// TIA Portal project "2025-26_Estampadora_Botonera_V17" (V17)

(* hardware
DEVICE "S7-1200 station_1"  S7-1200 Station
   slot 0: "Rack_0"  S7-1200 Rack  Rack  V1.0
   slot 1: "PLC_1"  CPU 1214C AC/DC/Rly  6ES7 214-1BG40-0XB0  V4.5
   slot 3: "AQ 1x12BIT_1"  AQ1 signal board  6ES7 232-4HA30-0XB0  V1.0
DEVICE "HMI_1"  KTP700 Basic PN
   slot 0: "HMI_1"  KTP700 Basic PN  6AV2 123-2GB03-0AX0  17.0.0.0
   slot 1: "HMI_RT_1"  KTP700 Basic PN  6AV2 123-2GB03-0AX0  17.0.0.0
   slot 5: "HMI_1.IE_CP_1"  PROFINET Interface  17.0.0.0
      slot 1: "PROFINET Interface_1"  PROFINET Interface
         slot 1: "Port_1"  Port
*)

// ===== PLC "PLC_1"  CPU 1214C AC/DC/Rly =====

VAR_GLOBAL   // PLC tag table "Tabla de variables estándar"
   "System_Byte" AT %MB1000 : Byte;
   "FirstScan" AT %M1000.0 : Bool;
   "DiagStatusUpdate" AT %M1000.1 : Bool;
   "AlwaysTRUE" AT %M1000.2 : Bool;
   "AlwaysFALSE" AT %M1000.3 : Bool;
   "INTERNA_Vacuna_libre" AT %M1001.0 : Bool;
   "INTERNA_Embalando_vacuna" AT %M1001.1 : Bool;
   "INTERNA_Soporte_libre" AT %M1001.2 : Bool;
   "INTERNA_Embalando_soporte" AT %M1001.3 : Bool;
   "INTERNA_Caja_libre" AT %M1001.4 : Bool;
   "INTERNA_Embalando_caja" AT %M1001.5 : Bool;
   "INTERNA_Robot_libre" AT %M1001.6 : Bool;
   "INTERNA_Robot_vacuna_hecho" AT %M1001.7 : Bool;
   "INTERNA_Robot_soporte_hecho" AT %M1002.0 : Bool;
   "OPCIN_sensor_caja_2" AT %I2.1 : Bool;
   "OPCIN_sensor_caja_1" AT %I2.0 : Bool;
   "OPCIN_sensor_caja_3" AT %I2.2 : Bool;
   "OPCIN_sensor_caja_A" AT %I2.3 : Bool;
   "OPCIN_sensor_caja_B" AT %I2.5 : Bool;
   "OPCIN_Emp_caja_A_front" AT %I3.1 : Bool;
   "OPCIN_Emp_caja_A_back" AT %I2.6 : Bool;
   "OPCIN_Emp_caja_B_front" AT %I2.7 : Bool;
   "OPCIN_Emp_caja_B_back" AT %I3.0 : Bool;
   "OPCOUT_Cinta_pre_caja" AT %Q2.0 : Bool;
   "OPCOUT_Cinta_post_caja" AT %Q2.1 : Bool;
   "OPCOUT_Cinta_alma_caja" AT %Q2.4 : Bool;
   "OPCOUT_Emp_caja_A" AT %Q2.2 : Bool;
   "OPCOUT_Emp_caja_B" AT %Q2.3 : Bool;
   "OPCOUT_Cajas" AT %Q3.2 : Bool;
   "OPCIN_Sensor_soporte" AT %I1.0 : Bool;
   "OPCIN_Vision_soporte" AT %IW34 : Int;
   "OPCIN_Sensor_soporte_A" AT %I1.2 : Bool;
   "OPCIN_Sensor_soporte_B" AT %I1.1 : Bool;
   "OPCIN_Emp_soporte_A_front" AT %I1.7 : Bool;
   "OPCIN_Emp_soporte_A_back" AT %I1.6 : Bool;
   "OPCIN_Emp_soporte_B_front" AT %I1.5 : Bool;
   "OPCIN_Emp_soporte_B_back" AT %I1.4 : Bool;
   "OPCOUT_Cinta_pre_soporte" AT %Q1.0 : Bool;
   "OPCOUT_Cinta_post_soporte" AT %Q1.1 : Bool;
   "OPCOUT_Cinta_alma_soporte" AT %Q1.5 : Bool;
   "OPCOUT_Cinta_curva_soporte" AT %Q1.4 : Bool;
   "OPCOUT_Soporte" AT %Q3.1 : Bool;
   "OPCOUT_Emp_soporte_A" AT %Q1.3 : Bool;
   "OPCOUT_Emp_soporte_B" AT %Q1.2 : Bool;
   "OPCIN_Sensor_vacuna" AT %I0.0 : Bool;
   "OPCIN_Vision_vacuna" AT %IW30 : Int;
   "OPCIN_Sensor_vacuna_A" AT %I0.2 : Bool;
   "OPCIN_Sensor_vacuna_B" AT %I0.1 : Bool;
   "OPCIN_Emp_vacuna_B_front" AT %I0.5 : Bool;
   "OPCIN_Emp_vacuna_B_back" AT %I0.4 : Bool;
   "OPCIN_Emp_vacuna_A_front" AT %I0.7 : Bool;
   "OPCIN_Emp_vacuna_A_back" AT %I0.6 : Bool;
   "OPCOUT_Cinta_pre_vacunas" AT %Q0.0 : Bool;
   "OPCOUT_Vacunas" AT %Q3.0 : Bool;
   "OPCOUT_Cinta_post_vacuna" AT %Q0.1 : Bool;
   "OPCOUT_Emp_vacuna_B" AT %Q0.2 : Bool;
   "OPCOUT_Emp_vacuna_A" AT %Q0.3 : Bool;
   "OPCOUT_Cinta_alma_vacuna" AT %Q0.5 : Bool;
   "OPCOUT_Cinta_curva_vacuna" AT %Q0.4 : Bool;
   "OPCIN_sensor_alma_soporte" AT %I1.3 : Bool;
   "OPCIN_sensor_alma_vacuna" AT %I0.3 : Bool;
   "OPCIN_sensor_alma_caja" AT %I2.4 : Bool;
   "OPCIN_PP_Rotating" AT %I3.5 : Bool;
   "OPCIN_PP_Moving_X" AT %I3.3 : Bool;
   "OPCIN_PP_Detected" AT %I3.2 : Bool;
   "OPCIN_PP_Moving_Z" AT %I3.4 : Bool;
   "OPCOUT_PP_CW" AT %Q3.4 : Bool;
   "OPCOUT_PP_CCW" AT %Q3.5 : Bool;
   "OPCOUT_PP_X" AT %Q3.6 : Bool;
   "OPCOUT_PP_Z" AT %Q3.7 : Bool;
   "OPCOUT_PP_Grab" AT %Q3.3 : Bool;
   "INTERNA_Robot_soporte" AT %M1002.1 : Bool;
   "INTERNA_Robot_vacuna" AT %M1002.2 : Bool;
   "CW_ROB1" AT %M1002.3 : Bool;
   "CW_ROB2" AT %M1002.4 : Bool;
   "CCW_ROB1" AT %M1002.5 : Bool;
   "CCW_ROB2" AT %M1002.6 : Bool;
   "GRAB_ROB1" AT %M1002.7 : Bool;
   "GRAB_ROB2" AT %M1003.0 : Bool;
   "X_ROB1" AT %M1003.1 : Bool;
   "X_ROB2" AT %M1003.2 : Bool;
   "Z_ROB1" AT %M1003.3 : Bool;
   "Z_ROB2" AT %M1003.4 : Bool;
   "CIN_ALMA_1" AT %M1003.5 : Bool;
   "CIN_ALMA_2" AT %M1003.6 : Bool;
   "Alarma_vacuna" AT %M1003.7 : Bool;
   "Alarma_soporte" AT %M1004.0 : Bool;
   "Alarma_caja" AT %M1004.1 : Bool;
   "BOOL_EMERGENCIA" AT %M1004.2 : Bool;
   "BOOL_REARME" AT %M1004.3 : Bool;
   "OPCIN_RESET" AT %I4.0 : Bool;
   "OPCIN_RESUME" AT %I4.1 : Bool;
   "OPCIN_SALIDA" AT %I4.2 : Bool;
   "OPCOUT_N_CICLOS" AT %QW30 : Int;
   "OPCIN_SETA" AT %I4.3 : Bool;
   "RESET" AT %M1004.4 : Bool;
   "RESUME" AT %M1004.5 : Bool;
   "FINAL" AT %M1004.6 : Bool;
   "SETA" AT %M1004.7 : Bool;
END_VAR

DATA_BLOCK "Llamadas_Robot_DB"   // DB4
{ S7_Optimized_Access := 'TRUE' }
VERSION : 0.1
// stored: InstanceOfName HANDLER
"HANDLER"
BEGIN
END_DATA_BLOCK

DATA_BLOCK "DATOS_HMI"   // DB18
{ S7_Optimized_Access := 'TRUE' }
VERSION : 0.1
   VAR
      Boton_Reset : Bool;
      Boton_Resume : Bool;
      Estado_Alarma : Bool;
      Estado_Vacuna : Int;
      Estado_Soporte : Int;
      Estado_Caja : Int;
      Estado_Embalaje : Int;
      "CAJAS TOTALES" : Int;
      "SETA EMERGENCIA" : Bool;
      "BOTON REARME" : Bool;
      "FIN DE PISTA" : Bool;
   END_VAR
BEGIN
END_DATA_BLOCK

DATA_BLOCK "EMERGENCIA_DB"   // DB19
{ S7_Optimized_Access := 'TRUE' }
VERSION : 0.1
// stored: InstanceOfName EMERGENCIA
"EMERGENCIA"
BEGIN
END_DATA_BLOCK

DATA_BLOCK "Cinta_Vacunas_DB"   // DB34
{ S7_Optimized_Access := 'TRUE' }
VERSION : 0.1
// stored: InstanceOfName Cinta_Vacunas
"Cinta_Vacunas"
BEGIN
END_DATA_BLOCK

DATA_BLOCK "Cinta_Vacunas_DB_1"   // DB49
{ S7_Optimized_Access := 'TRUE' }
VERSION : 0.1
// stored: InstanceOfName Cinta_Vacunas
"Cinta_Vacunas"
BEGIN
END_DATA_BLOCK

DATA_BLOCK "Cinta_soporte_DB"   // DB50
{ S7_Optimized_Access := 'TRUE' }
VERSION : 0.1
// stored: InstanceOfName Cinta_soporte
"Cinta_soporte"
BEGIN
END_DATA_BLOCK

DATA_BLOCK "Cinta_soporte_DB_1"   // DB51
{ S7_Optimized_Access := 'TRUE' }
VERSION : 0.1
// stored: InstanceOfName Cinta_soporte
"Cinta_soporte"
BEGIN
END_DATA_BLOCK

DATA_BLOCK "Cinta_cajas_DB"   // DB52
{ S7_Optimized_Access := 'TRUE' }
VERSION : 0.1
// stored: InstanceOfName Cinta_cajas
"Cinta_cajas"
BEGIN
END_DATA_BLOCK

DATA_BLOCK "Embalaje_DB"   // DB53
{ S7_Optimized_Access := 'TRUE' }
VERSION : 0.1
// stored: InstanceOfName Embalaje
"Embalaje"
BEGIN
END_DATA_BLOCK

DATA_BLOCK "Robot_Vacuna_DB"   // DB54
{ S7_Optimized_Access := 'TRUE' }
VERSION : 0.1
// stored: InstanceOfName Robot_Vacuna
"Robot_Vacuna"
BEGIN
END_DATA_BLOCK

DATA_BLOCK "Robot_Soporte_DB"   // DB55
{ S7_Optimized_Access := 'TRUE' }
VERSION : 0.1
// stored: InstanceOfName Robot_Soporte
"Robot_Soporte"
BEGIN
END_DATA_BLOCK

// folder: System blocks/Program resources

DATA_BLOCK "2s/X41"   // DB1
{ S7_Optimized_Access := 'TRUE' }
AUTHOR : Simatic
FAMILY : IEC
NAME : IEC_TMR
VERSION : 1.0
// stored: InstanceOfName IEC_TIMER
"IEC_TIMER"
BEGIN
END_DATA_BLOCK

DATA_BLOCK "2s/x42"   // DB2
{ S7_Optimized_Access := 'TRUE' }
AUTHOR : Simatic
FAMILY : IEC
NAME : IEC_TMR
VERSION : 1.0
// stored: InstanceOfName IEC_TIMER
"IEC_TIMER"
BEGIN
END_DATA_BLOCK

DATA_BLOCK "2s/X34"   // DB3
{ S7_Optimized_Access := 'TRUE' }
AUTHOR : Simatic
FAMILY : IEC
NAME : IEC_TMR
VERSION : 1.0
// stored: InstanceOfName IEC_TIMER
"IEC_TIMER"
BEGIN
END_DATA_BLOCK

DATA_BLOCK "T_Alarma_2"   // DB5
{ S7_Optimized_Access := 'TRUE' }
AUTHOR : Simatic
FAMILY : IEC
NAME : IEC_TMR
VERSION : 1.0
// stored: InstanceOfName IEC_TIMER
"IEC_TIMER"
BEGIN
END_DATA_BLOCK

DATA_BLOCK "T_Alarma_5"   // DB6
{ S7_Optimized_Access := 'TRUE' }
AUTHOR : Simatic
FAMILY : IEC
NAME : IEC_TMR
VERSION : 1.0
// stored: InstanceOfName IEC_TIMER
"IEC_TIMER"
BEGIN
END_DATA_BLOCK

DATA_BLOCK "T_Alarma_7"   // DB7
{ S7_Optimized_Access := 'TRUE' }
AUTHOR : Simatic
FAMILY : IEC
NAME : IEC_TMR
VERSION : 1.0
// stored: InstanceOfName IEC_TIMER
"IEC_TIMER"
BEGIN
END_DATA_BLOCK

DATA_BLOCK "T_Alarma_7_PRIMA"   // DB8
{ S7_Optimized_Access := 'TRUE' }
AUTHOR : Simatic
FAMILY : IEC
NAME : IEC_TMR
VERSION : 1.0
// stored: InstanceOfName IEC_TIMER
"IEC_TIMER"
BEGIN
END_DATA_BLOCK

DATA_BLOCK "T_Alarma_3"   // DB9
{ S7_Optimized_Access := 'TRUE' }
AUTHOR : Simatic
FAMILY : IEC
NAME : IEC_TMR
VERSION : 1.0
// stored: InstanceOfName IEC_TIMER
"IEC_TIMER"
BEGIN
END_DATA_BLOCK

DATA_BLOCK "T_alarma_6"   // DB10
{ S7_Optimized_Access := 'TRUE' }
AUTHOR : Simatic
FAMILY : IEC
NAME : IEC_TMR
VERSION : 1.0
// stored: InstanceOfName IEC_TIMER
"IEC_TIMER"
BEGIN
END_DATA_BLOCK

DATA_BLOCK "T_Alarma_9"   // DB11
{ S7_Optimized_Access := 'TRUE' }
AUTHOR : Simatic
FAMILY : IEC
NAME : IEC_TMR
VERSION : 1.0
// stored: InstanceOfName IEC_TIMER
"IEC_TIMER"
BEGIN
END_DATA_BLOCK

DATA_BLOCK "T_Alarma_9_PRIMA"   // DB12
{ S7_Optimized_Access := 'TRUE' }
AUTHOR : Simatic
FAMILY : IEC
NAME : IEC_TMR
VERSION : 1.0
// stored: InstanceOfName IEC_TIMER
"IEC_TIMER"
BEGIN
END_DATA_BLOCK

DATA_BLOCK "TIMER_ALARMA_FRESADORA"   // DB13
{ S7_Optimized_Access := 'TRUE' }
AUTHOR : Simatic
FAMILY : IEC
NAME : IEC_TMR
VERSION : 1.0
// stored: InstanceOfName IEC_TIMER
"IEC_TIMER"
BEGIN
END_DATA_BLOCK

DATA_BLOCK "T_alarma_1"   // DB14
{ S7_Optimized_Access := 'TRUE' }
AUTHOR : Simatic
FAMILY : IEC
NAME : IEC_TMR
VERSION : 1.0
// stored: InstanceOfName IEC_TIMER
"IEC_TIMER"
BEGIN
END_DATA_BLOCK

DATA_BLOCK "T_alarma_4"   // DB15
{ S7_Optimized_Access := 'TRUE' }
AUTHOR : Simatic
FAMILY : IEC
NAME : IEC_TMR
VERSION : 1.0
// stored: InstanceOfName IEC_TIMER
"IEC_TIMER"
BEGIN
END_DATA_BLOCK

DATA_BLOCK "T_alarma_8"   // DB16
{ S7_Optimized_Access := 'TRUE' }
AUTHOR : Simatic
FAMILY : IEC
NAME : IEC_TMR
VERSION : 1.0
// stored: InstanceOfName IEC_TIMER
"IEC_TIMER"
BEGIN
END_DATA_BLOCK

DATA_BLOCK "T_alarma_8_PRIMA"   // DB17
{ S7_Optimized_Access := 'TRUE' }
AUTHOR : Simatic
FAMILY : IEC
NAME : IEC_TMR
VERSION : 1.0
// stored: InstanceOfName IEC_TIMER
"IEC_TIMER"
BEGIN
END_DATA_BLOCK

DATA_BLOCK "1S/X411"   // DB20
{ S7_Optimized_Access := 'TRUE' }
AUTHOR : Simatic
FAMILY : IEC
NAME : IEC_TMR
VERSION : 1.0
// stored: InstanceOfName IEC_TIMER
"IEC_TIMER"
BEGIN
END_DATA_BLOCK

DATA_BLOCK "Timer_1s_X04A"   // DB21
{ S7_Optimized_Access := 'TRUE' }
AUTHOR : Simatic
FAMILY : IEC
NAME : IEC_TMR
VERSION : 1.0
// stored: InstanceOfName IEC_TIMER
"IEC_TIMER"
BEGIN
END_DATA_BLOCK

DATA_BLOCK "Timer_1s_X03"   // DB22
{ S7_Optimized_Access := 'TRUE' }
AUTHOR : Simatic
FAMILY : IEC
NAME : IEC_TMR
VERSION : 1.0
// stored: InstanceOfName IEC_TIMER
"IEC_TIMER"
BEGIN
END_DATA_BLOCK

DATA_BLOCK "Timer_1s_X130A"   // DB23
{ S7_Optimized_Access := 'TRUE' }
AUTHOR : Simatic
FAMILY : IEC
NAME : IEC_TMR
VERSION : 1.0
// stored: InstanceOfName IEC_TIMER
"IEC_TIMER"
BEGIN
END_DATA_BLOCK

DATA_BLOCK "Timer_1s_X130B"   // DB24
{ S7_Optimized_Access := 'TRUE' }
AUTHOR : Simatic
FAMILY : IEC
NAME : IEC_TMR
VERSION : 1.0
// stored: InstanceOfName IEC_TIMER
"IEC_TIMER"
BEGIN
END_DATA_BLOCK

DATA_BLOCK "1s/X231A"   // DB25
{ S7_Optimized_Access := 'TRUE' }
AUTHOR : Simatic
FAMILY : IEC
NAME : IEC_TMR
VERSION : 1.0
// stored: InstanceOfName IEC_TIMER
"IEC_TIMER"
BEGIN
END_DATA_BLOCK

DATA_BLOCK "1s/X230B"   // DB26
{ S7_Optimized_Access := 'TRUE' }
AUTHOR : Simatic
FAMILY : IEC
NAME : IEC_TMR
VERSION : 1.0
// stored: InstanceOfName IEC_TIMER
"IEC_TIMER"
BEGIN
END_DATA_BLOCK

DATA_BLOCK "1S/X230C"   // DB27
{ S7_Optimized_Access := 'TRUE' }
AUTHOR : Simatic
FAMILY : IEC
NAME : IEC_TMR
VERSION : 1.0
// stored: InstanceOfName IEC_TIMER
"IEC_TIMER"
BEGIN
END_DATA_BLOCK

DATA_BLOCK "3s/x37"   // DB28
{ S7_Optimized_Access := 'TRUE' }
AUTHOR : Simatic
FAMILY : IEC
NAME : IEC_TMR
VERSION : 1.0
// stored: InstanceOfName IEC_TIMER
"IEC_TIMER"
BEGIN
END_DATA_BLOCK

DATA_BLOCK "1s/X311B"   // DB29
{ S7_Optimized_Access := 'TRUE' }
AUTHOR : Simatic
FAMILY : IEC
NAME : IEC_TMR
VERSION : 1.0
// stored: InstanceOfName IEC_TIMER
"IEC_TIMER"
BEGIN
END_DATA_BLOCK

DATA_BLOCK "1s/X311C"   // DB30
{ S7_Optimized_Access := 'TRUE' }
AUTHOR : Simatic
FAMILY : IEC
NAME : IEC_TMR
VERSION : 1.0
// stored: InstanceOfName IEC_TIMER
"IEC_TIMER"
BEGIN
END_DATA_BLOCK

DATA_BLOCK "1s/X321A"   // DB31
{ S7_Optimized_Access := 'TRUE' }
AUTHOR : Simatic
FAMILY : IEC
NAME : IEC_TMR
VERSION : 1.0
// stored: InstanceOfName IEC_TIMER
"IEC_TIMER"
BEGIN
END_DATA_BLOCK

DATA_BLOCK "1S/X311"   // DB32
{ S7_Optimized_Access := 'TRUE' }
AUTHOR : Simatic
FAMILY : IEC
NAME : IEC_TMR
VERSION : 1.0
// stored: InstanceOfName IEC_TIMER
"IEC_TIMER"
BEGIN
END_DATA_BLOCK

DATA_BLOCK "1s/X39"   // DB33
{ S7_Optimized_Access := 'TRUE' }
AUTHOR : Simatic
FAMILY : IEC
NAME : IEC_TMR
VERSION : 1.0
// stored: InstanceOfName IEC_TIMER
"IEC_TIMER"
BEGIN
END_DATA_BLOCK

DATA_BLOCK "1s/X410"   // DB35
{ S7_Optimized_Access := 'TRUE' }
AUTHOR : Simatic
FAMILY : IEC
NAME : IEC_TMR
VERSION : 1.0
// stored: InstanceOfName IEC_TIMER
"IEC_TIMER"
BEGIN
END_DATA_BLOCK

DATA_BLOCK "1s/X44"   // DB36
{ S7_Optimized_Access := 'TRUE' }
AUTHOR : Simatic
FAMILY : IEC
NAME : IEC_TMR
VERSION : 1.0
// stored: InstanceOfName IEC_TIMER
"IEC_TIMER"
BEGIN
END_DATA_BLOCK

DATA_BLOCK "2s/X45"   // DB37
{ S7_Optimized_Access := 'TRUE' }
AUTHOR : Simatic
FAMILY : IEC
NAME : IEC_TMR
VERSION : 1.0
// stored: InstanceOfName IEC_TIMER
"IEC_TIMER"
BEGIN
END_DATA_BLOCK

DATA_BLOCK "2s/X46"   // DB38
{ S7_Optimized_Access := 'TRUE' }
AUTHOR : Simatic
FAMILY : IEC
NAME : IEC_TMR
VERSION : 1.0
// stored: InstanceOfName IEC_TIMER
"IEC_TIMER"
BEGIN
END_DATA_BLOCK

DATA_BLOCK "1s/X47"   // DB39
{ S7_Optimized_Access := 'TRUE' }
AUTHOR : Simatic
FAMILY : IEC
NAME : IEC_TMR
VERSION : 1.0
// stored: InstanceOfName IEC_TIMER
"IEC_TIMER"
BEGIN
END_DATA_BLOCK

DATA_BLOCK "1s/X48"   // DB40
{ S7_Optimized_Access := 'TRUE' }
AUTHOR : Simatic
FAMILY : IEC
NAME : IEC_TMR
VERSION : 1.0
// stored: InstanceOfName IEC_TIMER
"IEC_TIMER"
BEGIN
END_DATA_BLOCK

DATA_BLOCK "1s/X49"   // DB41
{ S7_Optimized_Access := 'TRUE' }
AUTHOR : Simatic
FAMILY : IEC
NAME : IEC_TMR
VERSION : 1.0
// stored: InstanceOfName IEC_TIMER
"IEC_TIMER"
BEGIN
END_DATA_BLOCK

DATA_BLOCK "1S/X511"   // DB42
{ S7_Optimized_Access := 'TRUE' }
AUTHOR : Simatic
FAMILY : IEC
NAME : IEC_TMR
VERSION : 1.0
// stored: InstanceOfName IEC_TIMER
"IEC_TIMER"
BEGIN
END_DATA_BLOCK

DATA_BLOCK "1S/X54"   // DB43
{ S7_Optimized_Access := 'TRUE' }
AUTHOR : Simatic
FAMILY : IEC
NAME : IEC_TMR
VERSION : 1.0
// stored: InstanceOfName IEC_TIMER
"IEC_TIMER"
BEGIN
END_DATA_BLOCK

DATA_BLOCK "2S/X55"   // DB44
{ S7_Optimized_Access := 'TRUE' }
AUTHOR : Simatic
FAMILY : IEC
NAME : IEC_TMR
VERSION : 1.0
// stored: InstanceOfName IEC_TIMER
"IEC_TIMER"
BEGIN
END_DATA_BLOCK

DATA_BLOCK "2S/X56"   // DB45
{ S7_Optimized_Access := 'TRUE' }
AUTHOR : Simatic
FAMILY : IEC
NAME : IEC_TMR
VERSION : 1.0
// stored: InstanceOfName IEC_TIMER
"IEC_TIMER"
BEGIN
END_DATA_BLOCK

DATA_BLOCK "2S/X57"   // DB46
{ S7_Optimized_Access := 'TRUE' }
AUTHOR : Simatic
FAMILY : IEC
NAME : IEC_TMR
VERSION : 1.0
// stored: InstanceOfName IEC_TIMER
"IEC_TIMER"
BEGIN
END_DATA_BLOCK

DATA_BLOCK "1S/X59"   // DB47
{ S7_Optimized_Access := 'TRUE' }
AUTHOR : Simatic
FAMILY : IEC
NAME : IEC_TMR
VERSION : 1.0
// stored: InstanceOfName IEC_TIMER
"IEC_TIMER"
BEGIN
END_DATA_BLOCK

DATA_BLOCK "2S/X510"   // DB48
{ S7_Optimized_Access := 'TRUE' }
AUTHOR : Simatic
FAMILY : IEC
NAME : IEC_TMR
VERSION : 1.0
// stored: InstanceOfName IEC_TIMER
"IEC_TIMER"
BEGIN
END_DATA_BLOCK

DATA_BLOCK "1S/X8.5"   // DB56
{ S7_Optimized_Access := 'TRUE' }
AUTHOR : Simatic
FAMILY : IEC
NAME : IEC_TMR
VERSION : 1.0
// stored: InstanceOfName IEC_TIMER
"IEC_TIMER"
BEGIN
END_DATA_BLOCK

DATA_BLOCK "XAUX"   // DB57
{ S7_Optimized_Access := 'TRUE' }
AUTHOR : Simatic
FAMILY : IEC
NAME : IEC_TMR
VERSION : 1.0
// stored: InstanceOfName IEC_TIMER
"IEC_TIMER"
BEGIN
END_DATA_BLOCK

DATA_BLOCK "2S/XAUX2"   // DB58
{ S7_Optimized_Access := 'TRUE' }
AUTHOR : Simatic
FAMILY : IEC
NAME : IEC_TMR
VERSION : 1.0
// stored: InstanceOfName IEC_TIMER
"IEC_TIMER"
BEGIN
END_DATA_BLOCK

DATA_BLOCK "1S/X412"   // DB59
{ S7_Optimized_Access := 'TRUE' }
AUTHOR : Simatic
FAMILY : IEC
NAME : IEC_TMR
VERSION : 1.0
// stored: InstanceOfName IEC_TIMER
"IEC_TIMER"
BEGIN
END_DATA_BLOCK

DATA_BLOCK "2S/X511"   // DB60
{ S7_Optimized_Access := 'TRUE' }
AUTHOR : Simatic
FAMILY : IEC
NAME : IEC_TMR
VERSION : 1.0
// stored: InstanceOfName IEC_TIMER
"IEC_TIMER"
BEGIN
END_DATA_BLOCK

DATA_BLOCK "2S/X512"   // DB61
{ S7_Optimized_Access := 'TRUE' }
AUTHOR : Simatic
FAMILY : IEC
NAME : IEC_TMR
VERSION : 1.0
// stored: InstanceOfName IEC_TIMER
"IEC_TIMER"
BEGIN
END_DATA_BLOCK

DATA_BLOCK "2S/X513"   // DB62
{ S7_Optimized_Access := 'TRUE' }
AUTHOR : Simatic
FAMILY : IEC
NAME : IEC_TMR
VERSION : 1.0
// stored: InstanceOfName IEC_TIMER
"IEC_TIMER"
BEGIN
END_DATA_BLOCK

DATA_BLOCK "2S/X514"   // DB63
{ S7_Optimized_Access := 'TRUE' }
AUTHOR : Simatic
FAMILY : IEC
NAME : IEC_TMR
VERSION : 1.0
// stored: InstanceOfName IEC_TIMER
"IEC_TIMER"
BEGIN
END_DATA_BLOCK

DATA_BLOCK "2S/X58"   // DB64
{ S7_Optimized_Access := 'TRUE' }
AUTHOR : Simatic
FAMILY : IEC
NAME : IEC_TMR
VERSION : 1.0
// stored: InstanceOfName IEC_TIMER
"IEC_TIMER"
BEGIN
END_DATA_BLOCK

DATA_BLOCK "2S/X52"   // DB65
{ S7_Optimized_Access := 'TRUE' }
AUTHOR : Simatic
FAMILY : IEC
NAME : IEC_TMR
VERSION : 1.0
// stored: InstanceOfName IEC_TIMER
"IEC_TIMER"
BEGIN
END_DATA_BLOCK

// folder: (top level)

FUNCTION_BLOCK "Embalaje"   // FB1, SCL
{ S7_Optimized_Access := 'TRUE' }
VERSION : 0.1
   VAR_INPUT
      sensor_alma_soporte : Bool;
      sensor_alma_vacuna : Bool;
      sensor_alma_caja_1 : Bool;
      Robot_libre : Bool;
      Robot_soporte_hecho : Bool;
      Robot_vacuna_hecho : Bool;
      N_soportes : Int := 1;
      N_vacunas : Int := 1;
      EMERGENCIA : Bool;
      REARME : Bool;
      "FIN DE PISTA" : Bool;
   END_VAR
   VAR_OUTPUT
      N_ESTADO : Int;
      Soporte_libre : Bool;
      Vacuna_libre : Bool;
      Embalando_soporte : Bool;
      Embalando_vacuna : Bool;
      Caja_libre : Bool;
      Embalando_caja : Bool;
      Robot_soporte : Bool;
      Robot_vacuna : Bool;
      Cinta_alma_caja : Bool;
      CAJAS_TOTALES : Int;
   END_VAR
   VAR
      Flanco_x35 : R_TRIG;
      Flanco_x36 : R_TRIG;
      Flanco_X37 : R_TRIG;
      Count_soportes : Int;
      Count_vacunas : Int;
      X30 : Bool;
      X310A : Bool;
      X310B : Bool;
      X311B : Bool;
      X310C : Bool;
      X311C : Bool;
      X320A : Bool;
      X321A : Bool;
      X320B : Bool;
      X33 : Bool;
      X34 : Bool;
      X35 : Bool;
      X36 : Bool;
      X37 : Bool;
      X38 : Bool;
      X39 : Bool;
      X310 : Bool;
      X311 : Bool;
      S30 : Bool;
      S310A : Bool;
      S310B : Bool;
      S311B : Bool;
      S310C : Bool;
      S311C : Bool;
      S320A : Bool;
      S321A : Bool;
      S320B : Bool;
      S33 : Bool;
      S34 : Bool;
      S35 : Bool;
      S36 : Bool;
      S37 : Bool;
      S38 : Bool;
      S39 : Bool;
      S310 : Bool;
      S311 : Bool;
   END_VAR
BEGIN
   "3s/x37".TON(IN:=#X37,
                PT:=T#3s);
   "1s/X311B".TON(IN:=#X311B,
                  PT:=T#1s);
   "1s/X311C".TON(IN:=#X311C,
                  PT:=T#1s);
   "1s/X321A".TON(IN:=#X321A,
                  PT:=T#1s);
   "1S/X311".TON(IN:=#X311,
                 PT:=T#1s);
   "1s/X39".TON(IN:=#X39,
                PT:=t#1s);
   "2s/X34".TON(IN:=#X34,
                PT:=T#2S);

   IF NOT #EMERGENCIA THEN
       //FUNCIONES DE TRANSICIÓN
       #S30 := (#X37 AND "3s/x37".Q) OR (#X311B) OR (#X311C) OR "FirstScan";
       IF NOT #"FIN DE PISTA" THEN
           #S310A := #X30 AND #sensor_alma_soporte AND #sensor_alma_vacuna;
           #S310B := #X30 AND NOT #sensor_alma_soporte;
           #S310C := #X30 AND NOT #sensor_alma_vacuna;
       ELSE
           #S310A := FALSE;
           #S310B := FALSE;
           #S310C := FALSE;
       END_IF;
       #S311B := #X310B AND #sensor_alma_soporte;
       #S311C := #X310C AND #sensor_alma_vacuna;
       #S320A := #X310A AND NOT #sensor_alma_caja_1;
       #S321A := #X320A AND #sensor_alma_caja_1;
       #S320B := #X320A AND #sensor_alma_caja_1;
       #S33 := (#X321A AND "1s/X321A".Q) OR #X320B;
       #S34 := (#X33 AND #Robot_libre) OR (#X311 AND "1S/X311".Q);
       #S35 := (#X34 AND #Robot_vacuna_hecho AND "2s/X34".Q) OR (#X39);
       #S36 := #X35 AND (#Count_vacunas >= #N_vacunas) AND #Robot_soporte_hecho;
       #S37 := #X36 AND (#Count_soportes >= #N_soportes);
       #S38 := #X35 AND (#Count_vacunas < #N_vacunas) AND #Robot_soporte_hecho;
       #S39 := #X38 AND #sensor_alma_vacuna;
       #S310 := #X36 AND (#Count_soportes < #N_soportes);
       #S311 := #X310 AND #sensor_alma_soporte;

       //FUNCIONES DE ACTIVACIÓN DE ETAPAS
       #X30 := #S30 OR #X30 AND NOT (#S310A OR #S310B OR #S310C);
       #X310A := #S310A OR #X310A AND NOT (#S320A OR #S320B);
       #X320A := #S320A OR #X320A AND NOT #S321A;
       #X321A := #S321A OR #X321A AND NOT #S33;
       #X320B := #S320B OR #X320B AND NOT #S33;
       #X310B := #S310B OR #X310B AND NOT #S311B;
       #X311B := #S311B OR #X311B AND NOT #S30;
       #X310C := #S310C OR #X310C AND NOT #S311C;
       #X311C := #S311C OR #X311C AND NOT #S30;
       #X33 := #S33 OR #X33 AND NOT #S34;
       #X34 := #S34 OR #X34 AND NOT #S35;
       #X35 := #S35 OR #X35 AND NOT (#S36 OR #S38);
       #X36 := #S36 OR #X36 AND NOT (#S37 OR #S39);
       #X37 := #S37 OR #X37 AND NOT #S30;
       #X38 := #S38 OR #X38 AND NOT #S39;
       #X39 := #S39 OR #X39 AND NOT #S35;
       #X310 := #S310 OR #X310 AND NOT #S311;
       #X311 := #S311 OR #X311 AND NOT #S34;



       //FUNCIONES DE SALIDA
       #Soporte_libre := #X310B OR #X310;
       #Vacuna_libre := #X310C OR #X38;
       #Embalando_soporte := #X311B OR #X311;
       #Embalando_vacuna := #X311C OR #X39;
       #Caja_libre := #X320A;
       #Embalando_caja := #X321A;
       #Robot_soporte := #X35;
       #Robot_vacuna := #X34;
       #Cinta_alma_caja := #X37; 
   ELSE
       #Soporte_libre := FALSE;
       #Vacuna_libre := FALSE;
       #Embalando_soporte := FALSE;
       #Embalando_vacuna := FALSE;
       #Caja_libre := FALSE;
       #Embalando_caja := FALSE;
       #Robot_soporte := FALSE;
       #Robot_vacuna := FALSE;
       #Cinta_alma_caja := FALSE;

   END_IF;

   IF #REARME THEN
       #X30 := TRUE;
       #X310A := FALSE;
       #X320A := FALSE;
       #X321A := FALSE;
       #X320B := FALSE;
       #X310B := FALSE;
       #X311B := FALSE;
       #X310C := FALSE;
       #X311C := FALSE;
       #X33 := FALSE;
       #X34 := FALSE;
       #X35 := FALSE;
       #X36 := FALSE;
       #X37 := FALSE;
       #X38 := FALSE;
       #X39 := FALSE;
       #X310 := FALSE;
       #X311 := FALSE;
   END_IF;

   IF #X30 OR #X310A OR #X320B THEN
       #N_ESTADO := 0;
   ELSIF #X310B OR #X311B THEN
       #N_ESTADO := 1;
   ELSIF #X310C OR #X311C THEN
       #N_ESTADO := 2;
   ELSIF #X320A OR #X321A THEN
       #N_ESTADO := 3;
   ELSIF #X33 THEN
       #N_ESTADO := 4;
   ELSIF #X34 THEN
       #N_ESTADO := 5;
   ELSIF #X35 THEN
       #N_ESTADO := 6;
   ELSIF #X38 OR #X39 THEN
       #N_ESTADO := 7;
   ELSIF #X36 THEN
       #N_ESTADO := 8;
   ELSIF #X310 OR #X311 THEN
       #N_ESTADO := 9;
   ELSIF #X37 THEN
       #N_ESTADO := 10;
   END_IF;





   //CONTADORES
   #Flanco_x35(CLK := #X35);
   IF #Flanco_x35.Q THEN
       #Count_vacunas := #Count_vacunas + 1;
   END_IF;
   #Flanco_x36(CLK := #X36);
   IF #Flanco_x36.Q THEN
       #Count_vacunas := 0;
       #Count_soportes := #Count_soportes + 1;
   END_IF;
   #Flanco_X37(CLK := #X37);
   IF #Flanco_X37.Q THEN
       #Count_soportes := 0;
       #CAJAS_TOTALES := #CAJAS_TOTALES + 1;
   END_IF;
END_FUNCTION_BLOCK

FUNCTION_BLOCK "Robot_Vacuna"   // FB2, SCL
{ S7_Optimized_Access := 'TRUE' }
VERSION : 0.1
   VAR_INPUT
      Robot_vacuna : Bool;
      PP_Rotating : Bool;
      PP_Moving_X : Bool;
      PP_Detected : Bool;
      EMERGENCIA : Bool;
      REARME : Bool;
   END_VAR
   VAR_OUTPUT
      PP_CW : Bool;
      PP_CCW : Bool;
      Robot_libre : Bool;
      PP_X : Bool;
      PP_Z : Bool;
      PP_Grab : Bool;
      Robot_vacuna_hecho : Bool;
   END_VAR
   VAR
      X40 : Bool;
      X41 : Bool;
      X42 : Bool;
      X43 : Bool;
      X44 : Bool;
      X45 : Bool;
      X46 : Bool;
      X47 : Bool;
      X48 : Bool;
      X49 : Bool;
      X410 : Bool;
      X411 : Bool;
      S40 : Bool;
      S41 : Bool;
      S42 : Bool;
      S43 : Bool;
      S44 : Bool;
      S45 : Bool;
      S46 : Bool;
      S47 : Bool;
      S48 : Bool;
      S49 : Bool;
      S410 : Bool;
      S411 : Bool;
      "X8,5" : Bool;
      "S8,5" : Bool;
      XAUX : Bool;
      SAUX : Bool;
      SAUX2 : Bool;
      XAUX2 : Bool;
      S412 : Bool;
      X412 : Bool;
   END_VAR
BEGIN
   "1s/X410".TON(IN:=#X410,
                 PT:=T#1s);
   "1s/X44".TON(IN:=#X44,
                PT:=T#2s);
   "2s/X45".TON(IN:=#X45,
                PT:=T#2s);
   "2s/X46".TON(IN:=#X46,
                PT:=T#2s);
   "1s/X47".TON(IN:=#X47,
                PT:=T#2s);
   "1s/X48".TON(IN:=#X48,
                PT:=T#2s);
   "1s/X49".TON(IN:=#X49,
                PT:=T#2s);
   "2s/X41".TON(IN:=#X41,
                PT:=T#2s);
   "2s/x42".TON(IN:=#X42,
                PT:=t#2s);
   "1S/X411".TON(IN:=#X411,
                   PT:=t#2s);

   "1S/X8.5".TON(IN:=#"X8,5",
                 PT:=T#2s);

   "XAUX".TON(IN:=#XAUX,
              PT:=T#2S);
   "2S/XAUX2".TON(IN:=#XAUX2,
                  PT:=T#2S);
   "1S/X412".TON(IN:=#X412,
                 PT:=T#1S);



   IF NOT #EMERGENCIA THEN
       //FUNCIONES DE TRANSICIÓN
       #S40 := (#X412 AND "1S/X412".Q) OR "FirstScan";
       #S41 := #X40 AND #Robot_vacuna;
       #S42 := #X41 AND "2s/X41".Q;(*

   *)
       #S43 := #X42 AND "2s/x42".Q;
       #S44 := #X43 AND #PP_Detected;
       #S45 := #X44 AND "1s/X44".Q;
       #S46 := #X45 AND "2s/X45".Q;
       #S47 := #X46 AND "2s/X46".Q;
       #S48 := #X47 AND "1s/X47".Q;
       #SAUX2 := #X48 AND "1s/X48".Q;
       #"S8,5" := #XAUX2 AND "2S/XAUX2".Q;
       #SAUX := #"X8,5" AND "1S/X8.5".Q;
       #S49 := #XAUX AND "XAUX".Q;
       #S410 := #X49 AND "1s/X49".Q;
       #S411:= #X410 AND "1s/X410".Q;
       #S412 := #X411 AND "1S/X411".Q;


       //FUNCIONES DE ACTIVACIÓN
       #X40 := #S40 OR #X40 AND NOT #S41;
       #X41 := #S41 OR #X41 AND NOT #S42;
       #X42 := #S42 OR #X42 AND NOT #S43;
       #X43 := #S43 OR #X43 AND NOT #S44;
       #X44 := #S44 OR #X44 AND NOT #S45;
       #X45 := #S45 OR #X45 AND NOT #S46;
       #X46 := #S46 OR #X46 AND NOT #S47;
       #X47 := #S47 OR #X47 AND NOT #S48;
       #X48 := #S48 OR #X48 AND NOT #SAUX2;
       #XAUX2 := #SAUX2 OR #XAUX2 AND NOT #"S8,5";
       #"X8,5" := #"S8,5" OR #"X8,5" AND NOT #SAUX;
       #XAUX := #SAUX OR #XAUX AND NOT #S49;
       #X49 := #S49 OR #X49 AND NOT #S410;
       #X410 := #S410 OR #X410 AND NOT #S411;
       #X411 := #S411 OR #X411 AND NOT #S412;
       #X412 := #S412 OR #X412 AND NOT #S40;


       //FUNCIONES DE SALIDA
       #Robot_libre := #X40;
       #PP_CW := #X47 OR #X48 OR #"X8,5";
       #PP_CCW := #X41 OR #X411;
       #PP_X := #X43 OR #X44 OR #X45 OR #X42 OR #X49 OR #X410;
       #PP_Z := #X43 OR #X44 OR #X410;
       #PP_Grab := #X44 OR #XAUX2 OR #X45 OR #X46 OR #X47 OR #X48 OR #X49 OR #X410 OR #"X8,5" OR #XAUX;
       #Robot_vacuna_hecho := #X412;
   ELSE
       #Robot_libre := FALSE;
       #PP_CW := FALSE;
       #PP_CCW := FALSE;
       #PP_X := FALSE;
       #PP_Z := FALSE;
       #PP_Grab := FALSE;
       #Robot_vacuna_hecho := FALSE;
   END_IF;

   IF #REARME THEN
       #X40 := TRUE;
       #X41 := FALSE;
       #X42 := FALSE;
       #X43 := FALSE;
       #X44 := FALSE;
       #X45 := FALSE;
       #X46 := FALSE;
       #X47 := FALSE;
       #X48 := FALSE;
       #X49 := FALSE;
       #X410 := FALSE;
   END_IF;
END_FUNCTION_BLOCK

FUNCTION_BLOCK "Robot_Soporte"   // FB3, SCL
{ S7_Optimized_Access := 'TRUE' }
VERSION : 0.1
   VAR_INPUT
      Robot_soporte : Bool;
      PP_Rotating : Bool;
      PP_Moving_X : Bool;
      PP_Detected : Bool;
      PP_Moving_Z : Bool;
      EMERGENCIA : Bool;
      REARME : Bool;
   END_VAR
   VAR_OUTPUT
      Robot_libre : Bool;
      PP_CW : Bool;
      PP_CCW : Bool;
      PP_X : Bool;
      PP_Z : Bool;
      PP_Grab : Bool;
      Robot_soporte_hecho : Bool;
   END_VAR
   VAR
      X50 : Bool;
      X51 : Bool;
      X52 : Bool;
      X53 : Bool;
      X54 : Bool;
      X55 : Bool;
      X56 : Bool;
      X57 : Bool;
      X58 : Bool;
      X59 : Bool;
      X510 : Bool;
      X511 : Bool;
      X512 : Bool;
      X513 : Bool;
      X514 : Bool;
      S50 : Bool;
      S51 : Bool;
      S52 : Bool;
      S53 : Bool;
      S54 : Bool;
      S55 : Bool;
      S56 : Bool;
      S57 : Bool;
      S58 : Bool;
      S59 : Bool;
      S510 : Bool;
      S511 : Bool;
      S512 : Bool;
      S513 : Bool;
      S514 : Bool;
   END_VAR
BEGIN
   "1S/X511".TON(IN:=#X511,
                 PT:=t#2s);
   "2S/X52".TON(IN:=#X52,
                PT:=T#2S);
   "1S/X54".TON(IN:=#X54,
                PT:=t#2s);
   "2S/X55".TON(IN:=#X55,
                PT:=t#2s);
   "2S/X56".TON(IN:=#X56,
                PT:=t#2s);
   "2S/X57".TON(IN:=#X57,
                PT:=t#2s);
   "2S/X58".TON(IN:=#X58,
                PT:=T#1S);
   "1S/X59".TON(IN:=#X59,
                PT:=t#2s);
   "2S/X510".TON(IN:=#X510,
                 PT:=t#2s);
   "2S/X511".TON(IN:=#X511,
                 PT:=T#1S);
   "2S/X512".TON(IN:=#X512,
                 PT:=T#1S);
   "2S/X513".TON(IN:=#X513,
                 PT:=T#2S);
   "2S/X514".TON(IN:=#X514,
                 PT:=T#2S);


   IF NOT #EMERGENCIA THEN
       //FUNCIONES DE TRANSICIÓN
       #S50 := (#X514 AND "2S/X514".Q) OR "FirstScan";
       #S51 := #X50 AND #Robot_soporte;
       #S52 := #X51 AND #PP_Rotating;
       #S53 := #X52 AND "2S/X52".Q;
       #S54 := #X53 AND #PP_Detected;
       #S55 := #X54 AND "1S/X54".Q;
       #S56 := #X55 AND "2S/X55".Q;
       #S57 := #X56 AND "2S/X56".Q;
       #S58 := #X57 AND "2S/X57".Q;
       #S59 := #X58 AND "2S/X58".Q;
       #S510 := #X59 AND "1S/X59".Q;
       #S511 := #X510 AND "2S/X510".Q;
       #S512 := #X511 AND "2S/X511".Q;
       #S513 := #X512 AND "2S/X512".Q;
       #S514 := #X513 AND "2S/X513".Q;

       //FUNCIONES DE ACTIVACIÓN
       #X50 := #S50 OR #X50 AND NOT #S51;
       #X51 := #S51 OR #X51 AND NOT #S52;
       #X52 := #S52 OR #X52 AND NOT #S53;
       #X53 := #S53 OR #X53 AND NOT #S54;
       #X54 := #S54 OR #X54 AND NOT #S55;
       #X55 := #S55 OR #X55 AND NOT #S56;
       #X56 := #S56 OR #X56 AND NOT #S57;
       #X57 := #S57 OR #X57 AND NOT #S58;
       #X58 := #S58 OR #X58 AND NOT #S59;
       #X59 := #S59 OR #X59 AND NOT #S510;
       #X510 := #S510 OR #X510 AND NOT #S511;
       #X511 := #S511 OR #X511 AND NOT #S512;
       #X512 := #S512 OR #X512 AND NOT #S513;
       #X513 := #S513 OR #X513 AND NOT #S514;
       #X514 := #S514 OR #X514 AND NOT #S50;

       //FUNCIONES DE SALIDA
       #Robot_libre := #X50;
       #PP_CW := #X51 OR #X513;
       #PP_CCW := #X57 OR #X59;
       #PP_X := #X52 OR #X53 OR #X54 OR #X55;
       #PP_Z := #X53 OR #X54 OR #X510 OR #X511;
       #PP_Grab := #X55 OR #X56 OR #X57 OR #X58 OR #X59 OR #X510 OR #X54;
       #Robot_soporte_hecho := #X514;
   ELSE
       #Robot_libre := FALSE;
       #PP_CW := FALSE;
       #PP_CCW := FALSE;
       #PP_X := FALSE;
       #PP_Z := FALSE;
       #PP_Grab := FALSE;
       #Robot_soporte_hecho := FALSE;
   END_IF;

   IF #REARME THEN
       #X50 := TRUE;
       #X51 := FALSE;
       #X52 := FALSE;
       #X53 := FALSE;
       #X54 := FALSE;
       #X55 := FALSE;
       #X56 := FALSE;
       #X57 := FALSE;
       #X58 := FALSE;
       #X59 := FALSE;
       #X510 := FALSE;
       #X511 := FALSE;
   END_IF;
END_FUNCTION_BLOCK

FUNCTION_BLOCK "HANDLER"   // FB4, SCL
{ S7_Optimized_Access := 'TRUE' }
VERSION : 0.1
   VAR_INPUT
      CCW_rob1 : Bool;
      CCW_rob2 : Bool;
      CW_rob1 : Bool;
      CW_rob2 : Bool;
      X_rob1 : Bool;
      X_rob2 : Bool;
      Z_rob1 : Bool;
      Z_rob2 : Bool;
      GRAB_rob1 : Bool;
      GRAB_rob2 : Bool;
      CIN_ALMA_1 : Bool;
      CIN_ALMA_2 : Bool;
      RESET_FISICO : Bool;
      RESUME_FISICO : Bool;
      FIN_PISTA_FISICO : Bool;
      SETA_FISICO : Bool;
      RESET_HMI : Bool;
      RESUME_HMI : Bool;
      FIN_HMI : Bool;
      SETA_HMI : Bool;
      N_HECHO : Int;
   END_VAR
   VAR_OUTPUT
      CCW : Bool;
      CW : Bool;
      Z : Bool;
      X : Bool;
      GRAB : Bool;
      CIN_ALMA : Bool;
      Alarma_general : Bool;
      RESET : Bool;
      RESUME : Bool;
      FINAL : Bool;
      SETA : Bool;
      N_HECHO_SALIDA : Int;
   END_VAR
   VAR
      AUX : Bool;
   END_VAR
BEGIN
   #CW := #CW_rob1 OR #CW_rob2;
   #CCW := #CCW_rob1 OR #CCW_rob2;
   #Z := #Z_rob1 OR #Z_rob2;
   #X := #X_rob1 OR #X_rob2;
   #GRAB := #GRAB_rob1 OR #GRAB_rob2;
   #CIN_ALMA := #CIN_ALMA_1 OR #CIN_ALMA_2;
   #Alarma_general := #FIN_PISTA_FISICO OR #RESET_FISICO OR #RESUME_FISICO;

   #AUX := NOT #SETA_FISICO;
   #RESET := #RESET_FISICO OR #RESET_HMI;
   #RESUME := #RESUME_FISICO OR #RESUME_HMI;
   #FINAL := #FIN_PISTA_FISICO OR #FIN_HMI;
   #SETA := #AUX OR #SETA_HMI;

   #N_HECHO_SALIDA := #N_HECHO;
END_FUNCTION_BLOCK

FUNCTION_BLOCK "EMERGENCIA"   // FB5, SCL
{ S7_Optimized_Access := 'TRUE' }
VERSION : 0.1
   VAR_INPUT
      SETA_EMERGENCIA : Bool;
      BOTON_REARME : Bool;
   END_VAR
   VAR_OUTPUT
      EMERGENCIA : Bool;
      REARME : Bool;
   END_VAR
   VAR
      X100 : Bool;
      X101 : Bool;
      X102 : Bool;
      X103 : Bool;
      S100 : Bool;
      S101 : Bool;
      S102 : Bool;
      S103 : Bool;
   END_VAR
BEGIN
   #S100 := #X103 OR "FirstScan";
   #S101 := #X100 AND #SETA_EMERGENCIA;
   #S102 := #X101 AND NOT #SETA_EMERGENCIA;
   #S103 := #X102 AND #BOTON_REARME;

   #X100 := #S100 OR #X100 AND NOT #S101;
   #X101 := #S101 OR #X101 AND NOT #S102;
   #X102 := #S102 OR #X102 AND NOT #S103;
   #X103 := #S103 OR #X103 AND NOT #S100;

   #EMERGENCIA := #X101 OR #X102;
   #REARME := #X103;
END_FUNCTION_BLOCK

FUNCTION_BLOCK "Cinta_Vacunas"   // FB7, SCL
{ S7_Optimized_Access := 'TRUE' }
VERSION : 0.1
   VAR_INPUT
      Sensor_vacuna : Bool;
      Vision_vacuna : Int;
      Sensor_vacuna_A : Bool;
      Sensor_vacuna_B : Bool;
      Emp_vacuna_B_front : Bool;
      Emp_vacuna_B_back : Bool;
      Emp_vacuna_A_front : Bool;
      Emp_vacuna_A_back : Bool;
      Vacuna_libre : Bool;
      Embalando_vacuna : Bool;
      RESET : Bool;
      RESUME : Bool;
      EMERGENCIA : Bool;
      REARME : Bool;
      "FIN DE PISTA" : Bool;
   END_VAR
   VAR_OUTPUT
      Cinta_pre_vacunas : Bool;
      Vacunas : Bool;
      Cinta_post_vacuna : Bool;
      Emp_vacuna_B : Bool;
      Emp_vacuna_A : Bool;
      Cinta_alma_vacuna : Bool;
      Cinta_curva_vacuna : Bool;
      ESTADO_ALARMA : Bool;
      N_ESTADO : Int;
   END_VAR
   VAR
      ID_Vacuna : Int;
      S01 : Bool;
      S02 : Bool;
      S03 : Bool;
      S04A : Bool;
      S04B : Bool;
      S041A : Bool;
      S041B : Bool;
      S042B : Bool;
      S05 : Bool;
      S06A : Bool;
      S06B : Bool;
      S061B : Bool;
      S07 : Bool;
      X01 : Bool;
      X02 : Bool;
      X03 : Bool;
      X04A : Bool;
      X04B : Bool;
      X041A : Bool;
      X041B : Bool;
      X042B : Bool;
      X05 : Bool;
      X06A : Bool;
      X06B : Bool;
      X061B : Bool;
      X07 : Bool;
      ALARMA : Bool;
   END_VAR
BEGIN
   "Timer_1s_X04A".TON(IN:=#X04A,
                       PT:=T#0.5s);
   "Timer_1s_X03".TON(IN:=#X03,
                      PT:=T#0.5s);

   IF #Vision_vacuna > 0 THEN
       #ID_Vacuna := #Vision_vacuna;
   END_IF;

   "T_Alarma_2".TON(IN:=#X03 AND NOT #ALARMA,
                    PT:=T#30s);
   "T_Alarma_5".TON(IN := #X02 AND NOT #ALARMA,
                    PT := T#30S);
   "T_Alarma_7".TON(IN := #X04B AND NOT #ALARMA,
                    PT := T#30s);
   "T_Alarma_7_PRIMA".TON(IN:=#X06B AND NOT #ALARMA,
                          PT:=T#30S);



   IF "T_Alarma_2".Q AND NOT #X05 THEN
       #ALARMA := TRUE;
   END_IF;
   IF "T_Alarma_5".Q AND NOT #X03 THEN
       #ALARMA := TRUE;
   END_IF;
   IF "T_Alarma_7".Q AND NOT #X041B THEN
       #ALARMA := TRUE;
   END_IF;
   IF "T_Alarma_7_PRIMA".Q AND NOT #X061B THEN
       #ALARMA := TRUE;
   END_IF;

   //ECUACIONES DE TRANSICION
   IF NOT #ALARMA AND NOT #EMERGENCIA THEN
       #S01 := (#X07 AND #Embalando_vacuna) OR (#X061B AND #Emp_vacuna_A_back) OR (#X042B AND #Emp_vacuna_B_back) OR "FirstScan";
       IF NOT #"FIN DE PISTA" THEN
           #S02 := #X01;
       ELSE
           #S02 := FALSE;
       END_IF;
       #S03 := #X02 AND #Sensor_vacuna;
       #S04A := #X03 AND (#ID_Vacuna <> 8);
       #S04B := #X03 AND (#ID_Vacuna = 8);
       #S041A := #X04A AND "Timer_1s_X04A".Q; // Condición de tiempo
       #S041B := #X04B AND #Sensor_vacuna_B;
       #S042B := #X041B AND #Emp_vacuna_B_front;
       #S05 := #X041A AND #Sensor_vacuna_A;
       #S06A := #X05 AND (#ID_Vacuna = 5);
       #S06B := #X05 AND (#ID_Vacuna <> 5);
       #S07 := #X06A AND #Vacuna_libre;
       #S061B := #X06B AND #Emp_vacuna_A_front;


       //ECUACIONES DE ACTIVACIÓN DE ETAPAS
       #X01 := #S01 OR #X01 AND NOT #S02;
       #X02 := #S02 OR #X02 AND NOT #S03;
       #X03 := #S03 OR #X03 AND NOT (#S04A OR #S04B); // Divergencia OR
       #X04A := #S04A OR #X04A AND NOT #S041A;
       #X041A := #S041A OR #X041A AND NOT #S05;
       #X04B := #S04B OR #X04B AND NOT #S041B;
       #X041B := #S041B OR #X041B AND NOT #S042B;
       #X042B := #S042B OR #X042B AND NOT #S01;   // Vuelta al inicio
       #X05 := #S05 OR #X05 AND NOT (#S06A OR #S06B); // Divergencia OR
       #X06A := #S06A OR #X06A AND NOT #S07;
       #X07 := #S07 OR #X07 AND NOT #S01;   // Vuelta al inicio
       #X06B := #S06B OR #X06B AND NOT #S061B;
       #X061B := #S061B OR #X061B AND NOT #S01;   // Vuelta al inicio


       //ACTIVACIÓN DE SALIDAS

       #Cinta_pre_vacunas := #X02 OR #X04A OR (#X04B AND "Timer_1s_X03".Q);
       #Vacunas := #X02;
       #Cinta_post_vacuna := #X041A OR #X04B OR #X07;
       #Emp_vacuna_B := #X041B;
       #Emp_vacuna_A := #X06B;
       #Cinta_curva_vacuna := #X07;
       #Cinta_alma_vacuna := #X07;

       //ESTADOS DEL PROCESO
       IF #X01 OR #X02 OR #X03 THEN
           #N_ESTADO := 1;
       ELSIF #X04B OR #X041B OR #X042B THEN
           #N_ESTADO := 2;
       ELSIF #X04A OR #X041A OR #X05 THEN
           #N_ESTADO := 3;
       ELSIF #X06B OR #X061B THEN
           #N_ESTADO := 4;
       ELSIF #X06A THEN
           #N_ESTADO := 5;
       ELSIF #X07 THEN
           #N_ESTADO := 6;
       END_IF;

   ELSE
       #Cinta_pre_vacunas := FALSE;
       #Vacunas := FALSE;
       #Cinta_post_vacuna := FALSE;
       #Emp_vacuna_B := FALSE;
       #Emp_vacuna_A := FALSE;
       #Cinta_curva_vacuna := FALSE;
       #Cinta_alma_vacuna := FALSE;
       #N_ESTADO := 0;
   END_IF;


   IF (#ALARMA AND #RESET) OR #REARME THEN
       #X01 := TRUE;
       #X02 := FALSE;
       #X03 := FALSE;
       #X04A := FALSE;
       #X041A := FALSE;
       #X04B := FALSE;
       #X041B := FALSE;
       #X042B := FALSE;
       #X05 := FALSE;
       #X06A := FALSE;
       #X07 := FALSE;
       #X06B := FALSE;
       #X061B := FALSE;
       #ALARMA := FALSE;
   ELSIF #ALARMA AND #RESUME THEN
       #ALARMA := FALSE;
   END_IF;
END_FUNCTION_BLOCK

FUNCTION_BLOCK "Cinta_soporte"   // FB8, SCL
{ S7_Optimized_Access := 'TRUE' }
VERSION : 0.1
   VAR_INPUT
      Sensor_soporte : Bool;
      Vision_soporte : Int;
      Sensor_soporte_A : Bool;
      Sensor_soporte_B : Bool;
      Emp_soporte_A_front : Bool;
      Emp_soporte_A_back : Bool;
      Emp_soporte_B_front : Bool;
      Emp_soporte_B_back : Bool;
      Soporte_libre : Bool;
      Embalando_soporte : Bool;
      RESET : Bool;
      RESUME : Bool;
      EMERGENCIA : Bool;
      REARME : Bool;
      "FIN DE PISTA" : Bool;
   END_VAR
   VAR_OUTPUT
      Cinta_pre_soporte : Bool;
      Cinta_post_soporte : Bool;
      Cinta_alma_soporte : Bool;
      Cinta_curva_soporte : Bool;
      Soporte : Bool;
      Emp_soporte_A : Bool;
      Emp_soporte_B : Bool;
      ALARMA : Bool;
      N_ESTADO : Int;
   END_VAR
   VAR
      ALARMA_1 : Bool;
      ID_Soporte : Int;
      S10 : Bool;
      S11 : Bool;
      S12 : Bool;
      S130A : Bool;
      S130B : Bool;
      S131A : Bool;
      S131B : Bool;
      S132B : Bool;
      S14 : Bool;
      S150A : Bool;
      S150B : Bool;
      S16 : Bool;
      S151B : Bool;
      X10 : Bool;
      X11 : Bool;
      X12 : Bool;
      X130A : Bool;
      X130B : Bool;
      X131B : Bool;
      X14 : Bool;
      X150A : Bool;
      X150B : Bool;
      X151B : Bool;
      X16 : Bool;
      X132B : Bool;
      X131A : Bool;
      Alarma_3 : Bool;
      Alarma_6 : Bool;
      Alarma_9 : Bool;
   END_VAR
BEGIN
   "Timer_1s_X130A".TON(IN:=#X130A,
                        PT:=T#0.5s);
   "Timer_1s_X130B".TON(IN:=#X130B,
                        PT:=T#0.5s);

   IF #Vision_soporte > 0 THEN
       #ID_Soporte := #Vision_soporte;
   END_IF;


   "T_Alarma_3".TON(IN:=#X12 AND NOT #ALARMA,
                    PT:=T#30S);
   "T_alarma_6".TON(IN:=#X11 AND NOT #ALARMA,
                    PT:=T#30S);
   "T_Alarma_9".TON(IN:=#X130B AND NOT #ALARMA,
                    PT:=T#30S);
   "T_Alarma_9_PRIMA".TON(IN:=#X12 AND NOT #ALARMA,
                          PT:=T#30S);



   IF "T_Alarma_3".Q AND NOT #X14 THEN
       #ALARMA := TRUE;
   END_IF;

   IF "T_alarma_6".Q AND NOT #X12 THEN
       #ALARMA := TRUE;
   END_IF;

   IF "T_Alarma_9".Q AND NOT #X131B THEN
       #ALARMA := TRUE;
   END_IF;

   IF "T_Alarma_9_PRIMA".Q AND (#ID_Soporte = 3) AND NOT #X14 THEN
       #ALARMA := TRUE;
   END_IF;

   //FUNCIONES DE ACTIVACION
   IF NOT #ALARMA AND NOT #EMERGENCIA THEN
       #S10 := (#X16 AND #Embalando_soporte) OR (#X151B AND #Emp_soporte_A_back) OR (#X132B AND #Emp_soporte_B_back) OR "FirstScan";
       IF NOT #"FIN DE PISTA" THEN
           #S11 := #X10;
       ELSE
           #S11 := FALSE;
       END_IF;
       #S12 := #X11 AND #Sensor_soporte;
       #S130A := #X12 AND (#ID_Soporte <> 9);
       #S130B := #X12 AND (#ID_Soporte = 9);
       #S131A := #X130A AND "Timer_1s_X130A".Q;
       #S131B := #X130B AND #Sensor_soporte_B;
       #S132B := #X131B AND #Emp_soporte_B_front;
       #S14 := #X131A AND #Sensor_soporte_A;
       #S150A := #X14 AND (#ID_Soporte = 6);
       #S150B := #X14 AND (#ID_Soporte <> 6);
       #S16 := #X150A AND #Soporte_libre;
       #S151B := #X150B AND #Emp_soporte_A_front;

       //FUNCIONES DE ACTIVACION DE ETAPAS
       #X10 := #S10 OR #X10 AND NOT #S11;
       #X11 := #S11 OR #X11 AND NOT #S12;
       #X12 := #S12 OR #X12 AND NOT (#S130A OR #S130B); // Divergencia OR
       #X130A := #S130A OR #X130A AND NOT #S131A;
       #X131A := #S131A OR #X131A AND NOT #S14;
       #X130B := #S130B OR #X130B AND NOT #S131B;
       #X131B := #S131B OR #X131B AND NOT #S132B;
       #X132B := #S132B OR #X132B AND NOT #S10;   // Vuelta al inicio
       #X14 := #S14 OR #X14 AND NOT (#S150A OR #S150B); // Divergencia OR
       #X150A := #S150A OR #X150A AND NOT #S16;
       #X16 := #S16 OR #X16 AND NOT #S10;   // Vuelta al inicio
       #X150B := #S150B OR #X150B AND NOT #S151B;
       #X151B := #S151B OR #X151B AND NOT #S10;   // Vuelta al inicio


       //FUNCIONES DE SALIDA
       #Cinta_pre_soporte := #X11 OR #X130A OR (#X130B AND "Timer_1s_X130B".Q);
       #Soporte := #X11;
       #Cinta_post_soporte := #X131A OR #X130B OR #X16;
       #Emp_soporte_B := #X131B;
       #Emp_soporte_A := #X150B;
       #Cinta_curva_soporte := #X16;
       #Cinta_alma_soporte := #X16;

       //ESTADOS DEL PROCESO
       IF #X11 OR #X12 THEN
           #N_ESTADO := 1;
       ELSIF #X130B OR #X131B OR #X132B THEN
           #N_ESTADO := 2;
       ELSIF #X130A OR #X131A OR #X14 THEN
           #N_ESTADO := 3;
       ELSIF #X150B OR #X151B THEN
           #N_ESTADO := 4;
       ELSIF #X150A THEN
           #N_ESTADO := 5;
       ELSIF #X16 THEN
           #N_ESTADO := 6;
       END_IF;
   ELSE
       #Cinta_pre_soporte := FALSE;
       #Soporte := FALSE;
       #Cinta_post_soporte := FALSE;
       #Emp_soporte_B := FALSE;
       #Emp_soporte_A := FALSE;
       #Cinta_curva_soporte := FALSE;
       #Cinta_alma_soporte := FALSE;
       #N_ESTADO := 0;
   END_IF;

   IF (#ALARMA AND #RESET) OR #REARME THEN
       #X10 := TRUE;
       #X11 := FALSE;
       #X12 := FALSE;
       #X130A := FALSE;
       #X131A := FALSE;
       #X130B := FALSE;
       #X131B := FALSE;
       #X132B := FALSE;
       #X14 := FALSE;
       #X150A := FALSE;
       #X16 := FALSE;
       #X150B := FALSE;
       #X151B := FALSE;
       #ALARMA := FALSE;
   ELSIF #ALARMA AND #RESUME THEN
       #ALARMA := FALSE;
   END_IF;
END_FUNCTION_BLOCK

FUNCTION_BLOCK "Cinta_cajas"   // FB9, SCL
{ S7_Optimized_Access := 'TRUE' }
VERSION : 0.1
   VAR_INPUT
      sensor_caja_2 : Bool;
      sensor_caja_1 : Bool;
      sensor_caja_3 : Bool;
      caja_libre : Bool;
      embalando_caja : Bool;
      sensor_caja_A : Bool;
      sensor_caja_B : Bool;
      Emp_caja_A_front : Bool;
      Emp_caja_A_back : Bool;
      Emp_caja_B_front : Bool;
      Emp_caja_B_back : Bool;
      RESET : Bool;
      RESUME : Bool;
      EMERGENCIA : Bool;
      REARME : Bool;
      "FIN DE PISTA" : Bool;
   END_VAR
   VAR_OUTPUT
      Cinta_pre_caja : Bool;
      Cinta_post_caja : Bool;
      Cinta_alma_caja : Bool;
      Emp_caja_A : Bool;
      Emp_caja_B : Bool;
      Cajas : Bool;
      Salida_alarma : Bool;
      N_ESTADO : Int;
   END_VAR
   VAR
      X20 : Bool;
      X21 : Bool;
      X22 : Bool;
      X230A : Bool;
      X231A : Bool;
      X232A : Bool;
      X230B : Bool;
      X231B : Bool;
      X232B : Bool;
      X233B : Bool;
      X230C : Bool;
      X231C : Bool;
      X232C : Bool;
      X233C : Bool;
      S20 : Bool;
      S21 : Bool;
      S22 : Bool;
      S230A : Bool;
      S231A : Bool;
      S232A : Bool;
      S230B : Bool;
      S231B : Bool;
      S232B : Bool;
      S233B : Bool;
      S230C : Bool;
      S231C : Bool;
      S232C : Bool;
      S233C : Bool;
      "1s/X231A" : TON_TIME;
      ALARMA : Bool;
   END_VAR
BEGIN
   "1s/X231A".TON(IN:=#X231A,
                  PT:=T#1s);

   "1s/X230B".TON(IN:=#X230B,
                  PT:=T#1s);
   "1S/X230C".TON(IN := #X230C,
                  PT := T#0.5s);


   "T_alarma_1".TON(IN:=#X232A AND NOT #ALARMA,
                    PT:=T#30S);
   "T_alarma_4".TON(IN := #X21 AND NOT #ALARMA,
                    PT := T#30S);
   "T_alarma_8".TON(IN:=#X231B AND NOT #ALARMA,
                    PT:=t#30s);
   "T_alarma_8_PRIMA".TON(IN:=#X231C AND NOT #ALARMA,
                          PT:=T#30S);


   //solo vuelve a x20 tras recibir embalando caja
   IF "T_alarma_1".Q AND NOT #X20 THEN
       #ALARMA := TRUE;
   END_IF;
   IF "T_alarma_4".Q AND NOT #X22 THEN
       #ALARMA := TRUE;
   END_IF;
   IF "T_alarma_8".Q AND NOT #X232B THEN
       #ALARMA := TRUE;
   END_IF;
   IF "T_alarma_8_PRIMA".Q AND NOT #X232C THEN
       #ALARMA := TRUE;
   END_IF;

   IF NOT #ALARMA AND NOT #EMERGENCIA THEN
       //FUNCIONES DE TRANSICIÓN
       #S20 := (#X232A AND "INTERNA_Embalando_caja") OR (#X233C AND #Emp_caja_A_back) OR (#X233B AND #Emp_caja_B_back) OR "FirstScan";
       IF NOT #"FIN DE PISTA" THEN
           #S21 := #X20;
       ELSE
           #S21 := False;
       END_IF;
       #S22 := #X21 AND #sensor_caja_2;
       #S230A := #X22 AND #sensor_caja_1 AND #sensor_caja_3;
       #S231A := #X230A AND "INTERNA_Caja_libre";
       #S232A := #X231A AND "1s/X231A".Q;
       #S230B := #X22 AND (NOT #sensor_caja_1) AND #sensor_caja_3;
       #S231B := #X230B AND "1s/X230B".Q;
       #S232B := #X231B AND #sensor_caja_B;
       #S233B := #X232B AND #Emp_caja_B_front;
       #S230C := #X22 AND NOT #sensor_caja_1 AND NOT #sensor_caja_3;
       #S231C := #X230C AND "1S/X230C".Q;
       #S232C := #X231C AND #sensor_caja_A;
       #S233C := #X232C AND #Emp_caja_A_front;

       //FUNCIONES DE ACTIVACIÓN DE ETAPAS
       #X20 := #S20 OR #X20 AND NOT #S21;
       #X21 := #S21 OR #X21 AND NOT #S22;
       #X22 := #S22 OR #X22 AND NOT (#S230A OR #S230B OR #S230C);
       #X230A := #S230A OR #X230A AND NOT #S231A;
       #X231A := #S231A OR #X231A AND NOT #S232A;
       #X232A := #S232A OR #X232A AND NOT #S20;
       #X230B := #S230B OR #X230B AND NOT #S231B;
       #X231B := #S231B OR #X231B AND NOT #S232B;
       #X232B := #S232B OR #X232B AND NOT #S233B;
       #X233B := #S233B OR #X233B AND NOT #S20;
       #X230C := #S230C OR #X230C AND NOT #S231C;
       #X231C := #S231C OR #X231C AND NOT #S232C;
       #X232C := #S232C OR #X232C AND NOT #S233C;
       #X233C := #S233C OR #X233C AND NOT #S20;

       //FUNCIONES DE SALIDA
       #Cinta_pre_caja := #X21 OR #X230B OR #X230C OR #X231A;
       #Cajas := #X21;
       #Cinta_post_caja := #X232A OR #X231B OR #X231C;
       #Emp_caja_B := #X232C;
       #Emp_caja_A := #X232B;
       #Cinta_alma_caja := #X232A;

       //ETAPAS DEL PROCESO
       IF #X20 OR #X21 OR #X22 THEN
           #N_ESTADO := 1;
       ELSIF #X230B OR #X231B OR #X232B OR #X233B THEN
           #N_ESTADO := 2;
       ELSIF #X230C OR #X231C OR #X232C OR #X233C THEN
           #N_ESTADO := 3;
       ELSIF #X230A THEN
           #N_ESTADO := 4;
       ELSIF #X231A OR #X232A THEN
           #N_ESTADO := 5;
       END_IF;


   ELSE
       #Cinta_pre_caja := FALSE;
       #Cajas := FALSE;
       #Cinta_post_caja := FALSE;
       #Emp_caja_B := FALSE;
       #Emp_caja_A := FALSE;
       #Cinta_alma_caja := FALSE;
       #N_ESTADO := 0;
   END_IF;


   IF (#ALARMA AND #RESET) OR #REARME THEN
       #X20 := TRUE;
       #X21 := FALSE;
       #X22 := FALSE;
       #X230A := FALSE;
       #X231A := FALSE;
       #X232A := FALSE;
       #X230B := FALSE;
       #X231B := FALSE;
       #X232B := FALSE;
       #X233B := FALSE;
       #X230C := FALSE;
       #X231C := FALSE;
       #X232C := FALSE;
       #X233C := FALSE;
       #ALARMA := FALSE;
   ELSIF #ALARMA AND #RESUME THEN
       #ALARMA := FALSE;
   END_IF;
END_FUNCTION_BLOCK

FUNCTION "MHJ-PLC-Lab-Function-S71200" : Void   // FC9000, SCL
{ S7_Optimized_Access := 'TRUE' }
VERSION : 0.1
   VAR_TEMP
      rdTimeReturn : Int;
      outputTime : DTL;
      SyncVal : Byte;
      forVal : Int;
      forVal_2 : Int;
      Value : Byte;
   END_VAR
   VAR CONSTANT
      CompVal : Byte := 16#34;
      Value_01 : Byte := 16#11;
      Value_01_DW : DWord := 16#A165_D992;
      Value_02_DW : DWord := 16#58BE_4401;
   END_VAR
BEGIN

   #Value:=PEEK(area := 16#82,
        dbNumber := 0,
        byteOffset := 511);
   #Value := #Value + 1;

   POKE(area := 16#82,
        dbNumber := 0,
        byteOffset := 511,
        value := #Value);

   POKE(area:=16#81,
        dbNumber:=0,
        byteOffset:=1016,
        value:=#Value_01_DW);
   POKE(area := 16#81,
        dbNumber := 0,
        byteOffset := 1020,
        value := #Value_02_DW);

   POKE(area := 16#81,
        dbNumber := 0,
        byteOffset := 511,
        value := B#16#00);

   FOR #forVal := 0 TO 120 DO
       FOR #forVal_2:=0 TO 10 DO
           #rdTimeReturn:=RD_SYS_T(#outputTime);
           #rdTimeReturn := WR_SYS_T(#outputTime);
           #rdTimeReturn := RD_SYS_T(#outputTime);
           #rdTimeReturn := WR_SYS_T(#outputTime);
       END_FOR;
       #SyncVal:= PEEK(area := 16#81,
                      dbNumber := 0,
                      byteOffset := 511);
       IF #SyncVal = #CompVal THEN
          GOTO M_1;
       END_IF;
   END_FOR;
   RETURN;

   M_1:
   POKE(area := 16#81,
        dbNumber := 0,
        byteOffset := 511,
        value := B#16#0);
END_FUNCTION

ORGANIZATION_BLOCK "Main"   // OB1, LAD, ProgramCycle
TITLE = "Main Program Sweep (Cycle)"
{ S7_Optimized_Access := 'TRUE' }
VERSION : 0.1
   VAR_INPUT
      Initial_Call : Bool;   // Initial call of this OB
      Remanence : Bool;   // =True, if remanent data are available
   END_VAR
BEGIN

REGION Network 1
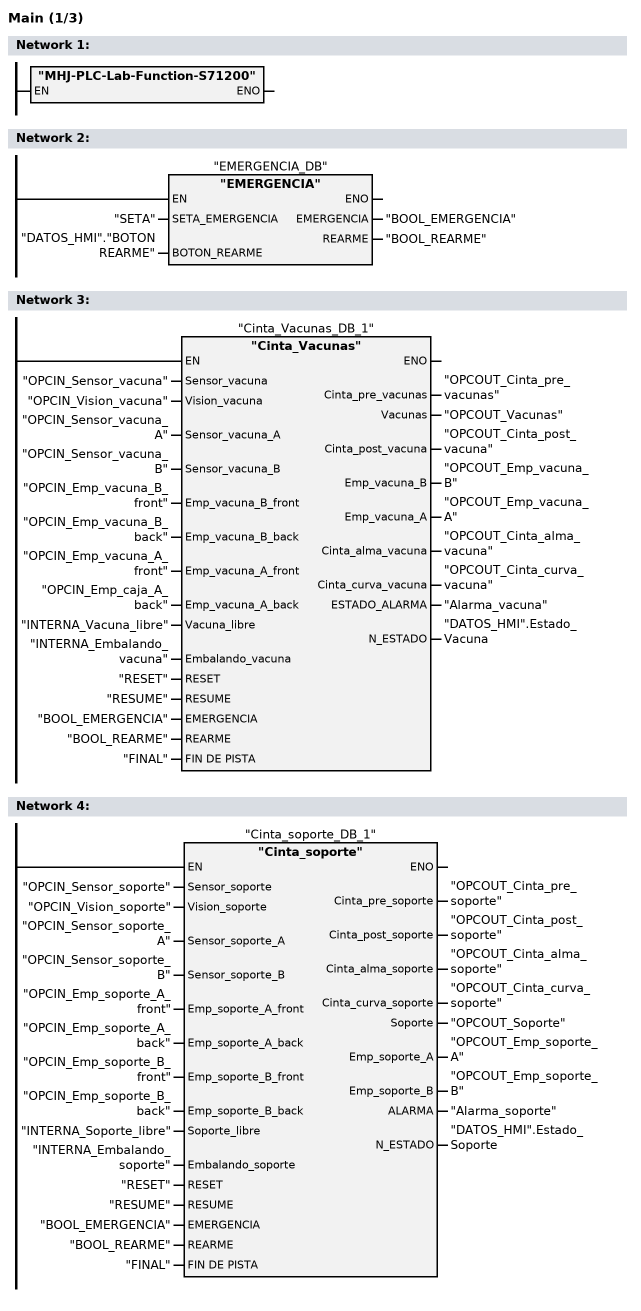
   RUNG wire#powerrail
      "MHJ-PLC-Lab-Function-S71200"()
   END_RUNG
   // the same network as SCL:
   "MHJ-PLC-Lab-Function-S71200"();
END_REGION

REGION Network 2
   RUNG wire#powerrail
      "EMERGENCIA_DB"(SETA_EMERGENCIA := "SETA", BOTON_REARME := "DATOS_HMI"."BOTON REARME", EMERGENCIA => "BOOL_EMERGENCIA", REARME => "BOOL_REARME")
   END_RUNG
   // the same network as SCL:
   "EMERGENCIA_DB"(SETA_EMERGENCIA := "SETA",   // "EMERGENCIA"
                   BOTON_REARME := "DATOS_HMI"."BOTON REARME",
                   EMERGENCIA => "BOOL_EMERGENCIA",
                   REARME => "BOOL_REARME");
END_REGION

REGION Network 3
   RUNG wire#powerrail
      "Cinta_Vacunas_DB_1"(Sensor_vacuna := "OPCIN_Sensor_vacuna", Vision_vacuna := "OPCIN_Vision_vacuna", Sensor_vacuna_A := "OPCIN_Sensor_vacuna_A", Sensor_vacuna_B := "OPCIN_Sensor_vacuna_B", Emp_vacuna_B_front := "OPCIN_Emp_vacuna_B_front", Emp_vacuna_B_back := "OPCIN_Emp_vacuna_B_back", Emp_vacuna_A_front := "OPCIN_Emp_vacuna_A_front", Emp_vacuna_A_back := "OPCIN_Emp_caja_A_back", Vacuna_libre := "INTERNA_Vacuna_libre", Embalando_vacuna := "INTERNA_Embalando_vacuna", RESET := "RESET", RESUME := "RESUME", EMERGENCIA := "BOOL_EMERGENCIA", REARME := "BOOL_REARME", "FIN DE PISTA" := "FINAL", Cinta_pre_vacunas => "OPCOUT_Cinta_pre_vacunas", Vacunas => "OPCOUT_Vacunas", Cinta_post_vacuna => "OPCOUT_Cinta_post_vacuna", Emp_vacuna_B => "OPCOUT_Emp_vacuna_B", Emp_vacuna_A => "OPCOUT_Emp_vacuna_A", Cinta_alma_vacuna => "OPCOUT_Cinta_alma_vacuna", Cinta_curva_vacuna => "OPCOUT_Cinta_curva_vacuna", ESTADO_ALARMA => "Alarma_vacuna", N_ESTADO => "DATOS_HMI".Estado_Vacuna)
   END_RUNG
   // the same network as SCL:
   "Cinta_Vacunas_DB_1"(Sensor_vacuna := "OPCIN_Sensor_vacuna",   // "Cinta_Vacunas"
                        Vision_vacuna := "OPCIN_Vision_vacuna",
                        Sensor_vacuna_A := "OPCIN_Sensor_vacuna_A",
                        Sensor_vacuna_B := "OPCIN_Sensor_vacuna_B",
                        Emp_vacuna_B_front := "OPCIN_Emp_vacuna_B_front",
                        Emp_vacuna_B_back := "OPCIN_Emp_vacuna_B_back",
                        Emp_vacuna_A_front := "OPCIN_Emp_vacuna_A_front",
                        Emp_vacuna_A_back := "OPCIN_Emp_caja_A_back",
                        Vacuna_libre := "INTERNA_Vacuna_libre",
                        Embalando_vacuna := "INTERNA_Embalando_vacuna",
                        RESET := "RESET",
                        RESUME := "RESUME",
                        EMERGENCIA := "BOOL_EMERGENCIA",
                        REARME := "BOOL_REARME",
                        "FIN DE PISTA" := "FINAL",
                        Cinta_pre_vacunas => "OPCOUT_Cinta_pre_vacunas",
                        Vacunas => "OPCOUT_Vacunas",
                        Cinta_post_vacuna => "OPCOUT_Cinta_post_vacuna",
                        Emp_vacuna_B => "OPCOUT_Emp_vacuna_B",
                        Emp_vacuna_A => "OPCOUT_Emp_vacuna_A",
                        Cinta_alma_vacuna => "OPCOUT_Cinta_alma_vacuna",
                        Cinta_curva_vacuna => "OPCOUT_Cinta_curva_vacuna",
                        ESTADO_ALARMA => "Alarma_vacuna",
                        N_ESTADO => "DATOS_HMI".Estado_Vacuna);
END_REGION

REGION Network 4
   RUNG wire#powerrail
      "Cinta_soporte_DB_1"(Sensor_soporte := "OPCIN_Sensor_soporte", Vision_soporte := "OPCIN_Vision_soporte", Sensor_soporte_A := "OPCIN_Sensor_soporte_A", Sensor_soporte_B := "OPCIN_Sensor_soporte_B", Emp_soporte_A_front := "OPCIN_Emp_soporte_A_front", Emp_soporte_A_back := "OPCIN_Emp_soporte_A_back", Emp_soporte_B_front := "OPCIN_Emp_soporte_B_front", Emp_soporte_B_back := "OPCIN_Emp_soporte_B_back", Soporte_libre := "INTERNA_Soporte_libre", Embalando_soporte := "INTERNA_Embalando_soporte", RESET := "RESET", RESUME := "RESUME", EMERGENCIA := "BOOL_EMERGENCIA", REARME := "BOOL_REARME", "FIN DE PISTA" := "FINAL", Cinta_pre_soporte => "OPCOUT_Cinta_pre_soporte", Cinta_post_soporte => "OPCOUT_Cinta_post_soporte", Cinta_alma_soporte => "OPCOUT_Cinta_alma_soporte", Cinta_curva_soporte => "OPCOUT_Cinta_curva_soporte", Soporte => "OPCOUT_Soporte", Emp_soporte_A => "OPCOUT_Emp_soporte_A", Emp_soporte_B => "OPCOUT_Emp_soporte_B", ALARMA => "Alarma_soporte", N_ESTADO => "DATOS_HMI".Estado_Soporte)
   END_RUNG
   // the same network as SCL:
   "Cinta_soporte_DB_1"(Sensor_soporte := "OPCIN_Sensor_soporte",   // "Cinta_soporte"
                        Vision_soporte := "OPCIN_Vision_soporte",
                        Sensor_soporte_A := "OPCIN_Sensor_soporte_A",
                        Sensor_soporte_B := "OPCIN_Sensor_soporte_B",
                        Emp_soporte_A_front := "OPCIN_Emp_soporte_A_front",
                        Emp_soporte_A_back := "OPCIN_Emp_soporte_A_back",
                        Emp_soporte_B_front := "OPCIN_Emp_soporte_B_front",
                        Emp_soporte_B_back := "OPCIN_Emp_soporte_B_back",
                        Soporte_libre := "INTERNA_Soporte_libre",
                        Embalando_soporte := "INTERNA_Embalando_soporte",
                        RESET := "RESET",
                        RESUME := "RESUME",
                        EMERGENCIA := "BOOL_EMERGENCIA",
                        REARME := "BOOL_REARME",
                        "FIN DE PISTA" := "FINAL",
                        Cinta_pre_soporte => "OPCOUT_Cinta_pre_soporte",
                        Cinta_post_soporte => "OPCOUT_Cinta_post_soporte",
                        Cinta_alma_soporte => "OPCOUT_Cinta_alma_soporte",
                        Cinta_curva_soporte => "OPCOUT_Cinta_curva_soporte",
                        Soporte => "OPCOUT_Soporte",
                        Emp_soporte_A => "OPCOUT_Emp_soporte_A",
                        Emp_soporte_B => "OPCOUT_Emp_soporte_B",
                        ALARMA => "Alarma_soporte",
                        N_ESTADO => "DATOS_HMI".Estado_Soporte);
END_REGION

REGION Network 5
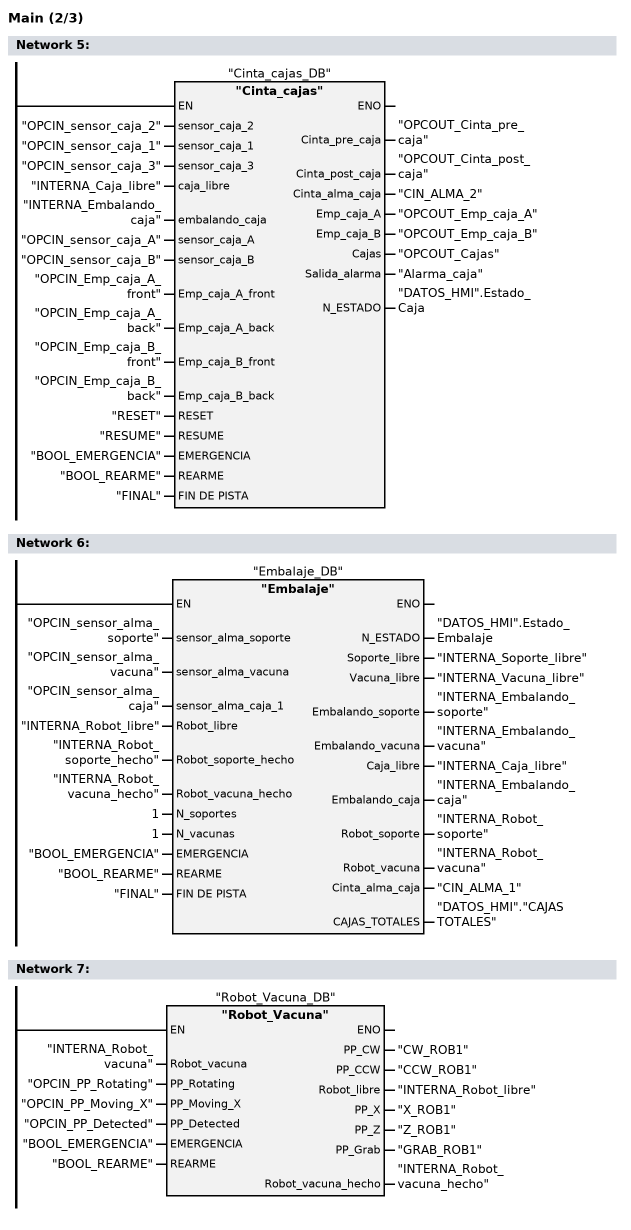
   RUNG wire#powerrail
      "Cinta_cajas_DB"(sensor_caja_2 := "OPCIN_sensor_caja_2", sensor_caja_1 := "OPCIN_sensor_caja_1", sensor_caja_3 := "OPCIN_sensor_caja_3", caja_libre := "INTERNA_Caja_libre", embalando_caja := "INTERNA_Embalando_caja", sensor_caja_A := "OPCIN_sensor_caja_A", sensor_caja_B := "OPCIN_sensor_caja_B", Emp_caja_A_front := "OPCIN_Emp_caja_A_front", Emp_caja_A_back := "OPCIN_Emp_caja_A_back", Emp_caja_B_front := "OPCIN_Emp_caja_B_front", Emp_caja_B_back := "OPCIN_Emp_caja_B_back", RESET := "RESET", RESUME := "RESUME", EMERGENCIA := "BOOL_EMERGENCIA", REARME := "BOOL_REARME", "FIN DE PISTA" := "FINAL", Cinta_pre_caja => "OPCOUT_Cinta_pre_caja", Cinta_post_caja => "OPCOUT_Cinta_post_caja", Cinta_alma_caja => "CIN_ALMA_2", Emp_caja_A => "OPCOUT_Emp_caja_A", Emp_caja_B => "OPCOUT_Emp_caja_B", Cajas => "OPCOUT_Cajas", Salida_alarma => "Alarma_caja", N_ESTADO => "DATOS_HMI".Estado_Caja)
   END_RUNG
   // the same network as SCL:
   "Cinta_cajas_DB"(sensor_caja_2 := "OPCIN_sensor_caja_2",   // "Cinta_cajas"
                    sensor_caja_1 := "OPCIN_sensor_caja_1",
                    sensor_caja_3 := "OPCIN_sensor_caja_3",
                    caja_libre := "INTERNA_Caja_libre",
                    embalando_caja := "INTERNA_Embalando_caja",
                    sensor_caja_A := "OPCIN_sensor_caja_A",
                    sensor_caja_B := "OPCIN_sensor_caja_B",
                    Emp_caja_A_front := "OPCIN_Emp_caja_A_front",
                    Emp_caja_A_back := "OPCIN_Emp_caja_A_back",
                    Emp_caja_B_front := "OPCIN_Emp_caja_B_front",
                    Emp_caja_B_back := "OPCIN_Emp_caja_B_back",
                    RESET := "RESET",
                    RESUME := "RESUME",
                    EMERGENCIA := "BOOL_EMERGENCIA",
                    REARME := "BOOL_REARME",
                    "FIN DE PISTA" := "FINAL",
                    Cinta_pre_caja => "OPCOUT_Cinta_pre_caja",
                    Cinta_post_caja => "OPCOUT_Cinta_post_caja",
                    Cinta_alma_caja => "CIN_ALMA_2",
                    Emp_caja_A => "OPCOUT_Emp_caja_A",
                    Emp_caja_B => "OPCOUT_Emp_caja_B",
                    Cajas => "OPCOUT_Cajas",
                    Salida_alarma => "Alarma_caja",
                    N_ESTADO => "DATOS_HMI".Estado_Caja);
END_REGION

REGION Network 6
   RUNG wire#powerrail
      "Embalaje_DB"(sensor_alma_soporte := "OPCIN_sensor_alma_soporte", sensor_alma_vacuna := "OPCIN_sensor_alma_vacuna", sensor_alma_caja_1 := "OPCIN_sensor_alma_caja", Robot_libre := "INTERNA_Robot_libre", Robot_soporte_hecho := "INTERNA_Robot_soporte_hecho", Robot_vacuna_hecho := "INTERNA_Robot_vacuna_hecho", N_soportes := 1, N_vacunas := 1, EMERGENCIA := "BOOL_EMERGENCIA", REARME := "BOOL_REARME", "FIN DE PISTA" := "FINAL", N_ESTADO => "DATOS_HMI".Estado_Embalaje, Soporte_libre => "INTERNA_Soporte_libre", Vacuna_libre => "INTERNA_Vacuna_libre", Embalando_soporte => "INTERNA_Embalando_soporte", Embalando_vacuna => "INTERNA_Embalando_vacuna", Caja_libre => "INTERNA_Caja_libre", Embalando_caja => "INTERNA_Embalando_caja", Robot_soporte => "INTERNA_Robot_soporte", Robot_vacuna => "INTERNA_Robot_vacuna", Cinta_alma_caja => "CIN_ALMA_1", CAJAS_TOTALES => "DATOS_HMI"."CAJAS TOTALES")
   END_RUNG
   // the same network as SCL:
   "Embalaje_DB"(sensor_alma_soporte := "OPCIN_sensor_alma_soporte",   // "Embalaje"
                 sensor_alma_vacuna := "OPCIN_sensor_alma_vacuna",
                 sensor_alma_caja_1 := "OPCIN_sensor_alma_caja",
                 Robot_libre := "INTERNA_Robot_libre",
                 Robot_soporte_hecho := "INTERNA_Robot_soporte_hecho",
                 Robot_vacuna_hecho := "INTERNA_Robot_vacuna_hecho",
                 N_soportes := 1,
                 N_vacunas := 1,
                 EMERGENCIA := "BOOL_EMERGENCIA",
                 REARME := "BOOL_REARME",
                 "FIN DE PISTA" := "FINAL",
                 N_ESTADO => "DATOS_HMI".Estado_Embalaje,
                 Soporte_libre => "INTERNA_Soporte_libre",
                 Vacuna_libre => "INTERNA_Vacuna_libre",
                 Embalando_soporte => "INTERNA_Embalando_soporte",
                 Embalando_vacuna => "INTERNA_Embalando_vacuna",
                 Caja_libre => "INTERNA_Caja_libre",
                 Embalando_caja => "INTERNA_Embalando_caja",
                 Robot_soporte => "INTERNA_Robot_soporte",
                 Robot_vacuna => "INTERNA_Robot_vacuna",
                 Cinta_alma_caja => "CIN_ALMA_1",
                 CAJAS_TOTALES => "DATOS_HMI"."CAJAS TOTALES");
END_REGION

REGION Network 7
   RUNG wire#powerrail
      "Robot_Vacuna_DB"(Robot_vacuna := "INTERNA_Robot_vacuna", PP_Rotating := "OPCIN_PP_Rotating", PP_Moving_X := "OPCIN_PP_Moving_X", PP_Detected := "OPCIN_PP_Detected", EMERGENCIA := "BOOL_EMERGENCIA", REARME := "BOOL_REARME", PP_CW => "CW_ROB1", PP_CCW => "CCW_ROB1", Robot_libre => "INTERNA_Robot_libre", PP_X => "X_ROB1", PP_Z => "Z_ROB1", PP_Grab => "GRAB_ROB1", Robot_vacuna_hecho => "INTERNA_Robot_vacuna_hecho")
   END_RUNG
   // the same network as SCL:
   "Robot_Vacuna_DB"(Robot_vacuna := "INTERNA_Robot_vacuna",   // "Robot_Vacuna"
                     PP_Rotating := "OPCIN_PP_Rotating",
                     PP_Moving_X := "OPCIN_PP_Moving_X",
                     PP_Detected := "OPCIN_PP_Detected",
                     EMERGENCIA := "BOOL_EMERGENCIA",
                     REARME := "BOOL_REARME",
                     PP_CW => "CW_ROB1",
                     PP_CCW => "CCW_ROB1",
                     Robot_libre => "INTERNA_Robot_libre",
                     PP_X => "X_ROB1",
                     PP_Z => "Z_ROB1",
                     PP_Grab => "GRAB_ROB1",
                     Robot_vacuna_hecho => "INTERNA_Robot_vacuna_hecho");
END_REGION

REGION Network 8
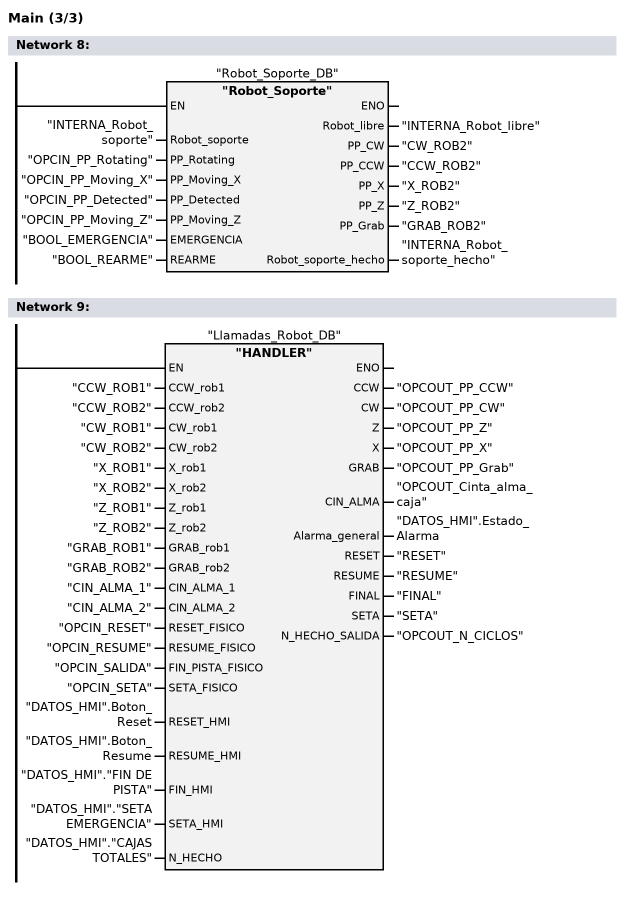
   RUNG wire#powerrail
      "Robot_Soporte_DB"(Robot_soporte := "INTERNA_Robot_soporte", PP_Rotating := "OPCIN_PP_Rotating", PP_Moving_X := "OPCIN_PP_Moving_X", PP_Detected := "OPCIN_PP_Detected", PP_Moving_Z := "OPCIN_PP_Moving_Z", EMERGENCIA := "BOOL_EMERGENCIA", REARME := "BOOL_REARME", Robot_libre => "INTERNA_Robot_libre", PP_CW => "CW_ROB2", PP_CCW => "CCW_ROB2", PP_X => "X_ROB2", PP_Z => "Z_ROB2", PP_Grab => "GRAB_ROB2", Robot_soporte_hecho => "INTERNA_Robot_soporte_hecho")
   END_RUNG
   // the same network as SCL:
   "Robot_Soporte_DB"(Robot_soporte := "INTERNA_Robot_soporte",   // "Robot_Soporte"
                      PP_Rotating := "OPCIN_PP_Rotating",
                      PP_Moving_X := "OPCIN_PP_Moving_X",
                      PP_Detected := "OPCIN_PP_Detected",
                      PP_Moving_Z := "OPCIN_PP_Moving_Z",
                      EMERGENCIA := "BOOL_EMERGENCIA",
                      REARME := "BOOL_REARME",
                      Robot_libre => "INTERNA_Robot_libre",
                      PP_CW => "CW_ROB2",
                      PP_CCW => "CCW_ROB2",
                      PP_X => "X_ROB2",
                      PP_Z => "Z_ROB2",
                      PP_Grab => "GRAB_ROB2",
                      Robot_soporte_hecho => "INTERNA_Robot_soporte_hecho");
END_REGION

REGION Network 9
   RUNG wire#powerrail
      "Llamadas_Robot_DB"(CCW_rob1 := "CCW_ROB1", CCW_rob2 := "CCW_ROB2", CW_rob1 := "CW_ROB1", CW_rob2 := "CW_ROB2", X_rob1 := "X_ROB1", X_rob2 := "X_ROB2", Z_rob1 := "Z_ROB1", Z_rob2 := "Z_ROB2", GRAB_rob1 := "GRAB_ROB1", GRAB_rob2 := "GRAB_ROB2", CIN_ALMA_1 := "CIN_ALMA_1", CIN_ALMA_2 := "CIN_ALMA_2", RESET_FISICO := "OPCIN_RESET", RESUME_FISICO := "OPCIN_RESUME", FIN_PISTA_FISICO := "OPCIN_SALIDA", SETA_FISICO := "OPCIN_SETA", RESET_HMI := "DATOS_HMI".Boton_Reset, RESUME_HMI := "DATOS_HMI".Boton_Resume, FIN_HMI := "DATOS_HMI"."FIN DE PISTA", SETA_HMI := "DATOS_HMI"."SETA EMERGENCIA", N_HECHO := "DATOS_HMI"."CAJAS TOTALES", CCW => "OPCOUT_PP_CCW", CW => "OPCOUT_PP_CW", Z => "OPCOUT_PP_Z", X => "OPCOUT_PP_X", GRAB => "OPCOUT_PP_Grab", CIN_ALMA => "OPCOUT_Cinta_alma_caja", Alarma_general => "DATOS_HMI".Estado_Alarma, RESET => "RESET", RESUME => "RESUME", FINAL => "FINAL", SETA => "SETA", N_HECHO_SALIDA => "OPCOUT_N_CICLOS")
   END_RUNG
   // the same network as SCL:
   "Llamadas_Robot_DB"(CCW_rob1 := "CCW_ROB1",   // "HANDLER"
                       CCW_rob2 := "CCW_ROB2",
                       CW_rob1 := "CW_ROB1",
                       CW_rob2 := "CW_ROB2",
                       X_rob1 := "X_ROB1",
                       X_rob2 := "X_ROB2",
                       Z_rob1 := "Z_ROB1",
                       Z_rob2 := "Z_ROB2",
                       GRAB_rob1 := "GRAB_ROB1",
                       GRAB_rob2 := "GRAB_ROB2",
                       CIN_ALMA_1 := "CIN_ALMA_1",
                       CIN_ALMA_2 := "CIN_ALMA_2",
                       RESET_FISICO := "OPCIN_RESET",
                       RESUME_FISICO := "OPCIN_RESUME",
                       FIN_PISTA_FISICO := "OPCIN_SALIDA",
                       SETA_FISICO := "OPCIN_SETA",
                       RESET_HMI := "DATOS_HMI".Boton_Reset,
                       RESUME_HMI := "DATOS_HMI".Boton_Resume,
                       FIN_HMI := "DATOS_HMI"."FIN DE PISTA",
                       SETA_HMI := "DATOS_HMI"."SETA EMERGENCIA",
                       N_HECHO := "DATOS_HMI"."CAJAS TOTALES",
                       CCW => "OPCOUT_PP_CCW",
                       CW => "OPCOUT_PP_CW",
                       Z => "OPCOUT_PP_Z",
                       X => "OPCOUT_PP_X",
                       GRAB => "OPCOUT_PP_Grab",
                       CIN_ALMA => "OPCOUT_Cinta_alma_caja",
                       Alarma_general => "DATOS_HMI".Estado_Alarma,
                       RESET => "RESET",
                       RESUME => "RESUME",
                       FINAL => "FINAL",
                       SETA => "SETA",
                       N_HECHO_SALIDA => "OPCOUT_N_CICLOS");
END_REGION
END_ORGANIZATION_BLOCK

(* ===== HMI "HMI_RT_1" =====
system functions are stored by id; their names below are inferred from use
connection "HMI_Connection_2": ETHERNET, SMART_S7_1200_OMS

HMI tags "Default tag table"
   "DATOS_HMI_Boton_Reset" : Bool = PLC DATOS_HMI.Boton_Reset, 1 s
   "DATOS_HMI_Boton_Resume" : Bool = PLC DATOS_HMI.Boton_Resume, 1 s
   "DATOS_HMI_Estado_Vacuna" : Int = PLC DATOS_HMI.Estado_Vacuna, 1 s
   "DATOS_HMI_Estado_Soporte" : Int = PLC DATOS_HMI.Estado_Soporte, 1 s
   "DATOS_HMI_Estado_Caja" : Int = PLC DATOS_HMI.Estado_Caja, 1 s
   "DATOS_HMI_Estado_Embalaje" : Int = PLC DATOS_HMI.Estado_Embalaje, 1 s
   "DATOS_HMI_CAJAS TOTALES" : Int = PLC DATOS_HMI."CAJAS TOTALES", 1 s
   "DATOS_HMI_SETA EMERGENCIA" : Bool = PLC DATOS_HMI."SETA EMERGENCIA", 1 s
   "DATOS_HMI_BOTON REARME" : Bool = PLC DATOS_HMI."BOTON REARME", 1 s
   "DATOS_HMI_FIN DE PISTA" : Bool = PLC DATOS_HMI."FIN DE PISTA", 1 s

text list "ESTADO_VACUNA": 0 'ALARMA'; 1 'DETECTADO TIPO DE VACUNA'; 2 'DESECHANDO LAS VACUNAS TIPO B'; 3 'MOVIENDO VACUNA AL SIGUIENTE PUNTO DE DECISIÓN'; 4 'DESECHANDO VACUNA INSERVIBLE'; 5 'ESPERANDO A QUE FALTE VACUNA'; 6 'ENTREGANDO VACUNA'

text list "ESTADO SOPORTE": 0 'ALARMA'; 1 'DETECTANDO TIPO DE SOPORTE'; 2 'DESECHANDO SOPORTE DE TIPO B'; 3 'MOVIENDO SOPORTE AL SIGUIENTE PUNTO DE DECISIÓN'; 4 'DESECHANDO SOPORTE INSERVIBLE'; 5 'ESPERANDO A QUE FALTEN SOPORTES'; 6 'ENTREGANDO SOPORTES'

text list "ESTADO CAJAS": 0 'ALARMA'; 1 'DECIDIENDO TIPO DE CAJA'; 2 'DESECHANDO CAJA TIPO B'; 3 'DESECHANDO CAJA INSERVIBLE'; 4 'ESPERANDO A QUE FALTE CAJA'; 5 'ENTREGANDO CAJA'

text list "ESTADO EMBALAJE": 0 'VALORANDO QUE FALTA PARA INICIAR EL PROCESO'; 1 'RECIBIENDO SOPORTE'; 2 'RECIBIENDO VACUNA'; 3 'RECIBIENDO CAJA'; 4 'ESPERANDO AL ROBOT'; 5 'ROBOT INTRODUCIENDO SOPORTE'; 6 'ROBOT INTRODUCIENDO VACUNA'; 7 'COMO NO HE ALCANZADO EL NUMERO DE VACUNAS POR SOPORTE, REPITO PROCESO'; 8 'VALORANDO SI HE INTRODUCIDO LOS SOPORTES POR CAJA NECESARIOS'; 9 'COMO NO HE ALCANZADO EL NUMERO DE SOPORTES POR CAJA, REPITO PROCESO'; 10 'ENTREGANDO CAJA LLENA'

Template "Template_1" 800x480
   Button "Exit" at 714,429 size 71x50; TextOff 'Exit'; PictureOff "ExitRuntime_KTP700_Basic_DP_TR"; PictureOn "ExitRuntime_KTP700_Basic_DP_TR"
      on Release: StopRuntime(0)
   Button "Template_Button" at 614,429 size 71x50; TextOff 'Text'
   Button "Template_Button_1" at 514,429 size 71x50; TextOff 'Text'
   Button "Template_Button_2" at 414,429 size 71x50; TextOff 'Text'
   Button "Template_Button_3" at 314,429 size 71x50; TextOff 'Text'
   Button "Template_Button_4" at 214,429 size 71x50; TextOff 'Text'
   Button "Alarms" at 114,429 size 71x50; TextOff 'Alarms'; PictureOff "AlarmDisplay_KTP700_Basic_DP_TR"; PictureOn "AlarmDisplay_KTP700_Basic_DP_TR"
      on Release: function_ef3f5d25("Alarm window_Unacknowledged", -1)
   Button "Start screen" at 14,429 size 71x50; TextOff 'Start screen'; PictureOff "NavigateHome_KTP700_Basic_DP_TR"; PictureOn "NavigateHome_KTP700_Basic_DP_TR"
      on Release: ActivateScreen("Root screen", 0)
   SymbolicIOField "Symbolic_IO_Field_Screen" at 93,9 size 600x33; TextOff '0'; TextOn '1'; TextList "TextList_ScreenNames"
   DateTimeField "HmiScreenItemData" at 695,25 size 105x25
   DateTimeField "HmiScreenItemData_1" at 695,0 size 105x25
   GraphicView "Logo" at 0,0 size 91x51; Picture "Logo of HMI_1"

screen "Root screen" 800x480, template "Template_1"
   Button "Button_1" at 95,83 size 131x68; TextOff 'ir a alarmas'
      on Click: ActivateScreen("alarmas", 0)
   Button "Button_2" at 704,389 size 96x32; TextOff 'volver'
      on Click: function_efd93a16()
   Button "Button_3" at 246,83 size 131x68; TextOff 'ir a estados'
      on Click: ActivateScreen("Informacion", 0)
   Button "Button_4" at 399,83 size 131x68; TextOff 'ir a emergencia'
      on Click: ActivateScreen("emergencia", 0)

screen "alarmas" 800x480
   Button "Button_1" at 180,85 size 229x183; TextOff 'reset'
      on Press: function_b14e0dd5("DATOS_HMI_Boton_Reset", 0)
   Button "Button_2" at 436,85 size 226x179; TextOff 'resume'
      on Press: function_b14e0dd5("DATOS_HMI_Boton_Resume", 0)
   Button "Button_3" at 704,448 size 96x32; TextOff 'volver'
      on Click: function_efd93a16()
   Button "Button_4" at 0,448 size 96x32; TextOff 'ir a home'
      on Click: ActivateScreen("Root screen", 0)
   Button "Button_5" at 180,280 size 484x69; TextOff 'TERMINAR CICLO'
      on Press: InvertBit("DATOS_HMI_FIN DE PISTA")

screen "Informacion" 800x480
   SymbolicIOField "Symbolic I/O field_1" at 403,66 size 371x82; TextOff '0'; TextOn '1'; TextList "ESTADO SOPORTE"
      ProcessValue <- "DATOS_HMI_Estado_Soporte"
   Button "Button_1" at 704,448 size 96x32; TextOff 'volver'
      on Click: function_efd93a16()
   Button "Button_2" at 0,448 size 96x32; TextOff 'ir a home'
      on Click: ActivateScreen("Root screen", 0)
   TextField "Text field_1" at 406,42 size 93x23; Text 'SOPORTES'
   SymbolicIOField "Symbolic I/O field_2" at 26,66 size 371x83; TextOn '1'; TextOff '0'; TextList "ESTADO_VACUNA"
      ProcessValue <- "DATOS_HMI_Estado_Vacuna"
   TextField "Text field_2" at 26,41 size 85x23; Text 'VACUNAS'
   SymbolicIOField "Symbolic I/O field_3" at 26,234 size 371x87; TextOn '1'; TextOff '0'; TextList "ESTADO CAJAS"
      ProcessValue <- "DATOS_HMI_Estado_Caja"
   TextField "Text field_3" at 26,209 size 58x23; Text 'CAJAS'
   SymbolicIOField "Symbolic I/O field_4" at 403,234 size 371x87; TextOn '1'; TextOff '0'; TextList "ESTADO EMBALAJE"
      ProcessValue <- "DATOS_HMI_Estado_Embalaje"
   TextField "Text field_4" at 403,209 size 91x23; Text 'EMBALAJE'
   IOField "I/O field_1" at 674,386 size 96x32; FormatPattern 9
      ProcessValue <- "DATOS_HMI_CAJAS TOTALES"
   TextField "Text field_5" at 493,389 size 181x23; Text 'CAJAS PROCESADAS:'

screen "emergencia" 800x480
   Button "Button_1" at 329,122 size 210x139; TextOff 'seta de emergencia'
      on Click: InvertBit("DATOS_HMI_SETA EMERGENCIA")
   Button "Button_2" at 332,282 size 206x32; TextOff 'rearme'
      on Press: function_b14e0dd5("DATOS_HMI_BOTON REARME", 0)
   Button "Button_3" at 704,448 size 96x32; TextOff 'volver'
      on Click: function_efd93a16()
   Button "Button_4" at 0,448 size 96x32; TextOff 'ir a home'
      on Click: ActivateScreen("Root screen", 0)
*)